FUNCTION_BLOCK "FB40_CommSlave"
{ S7_Optimized_Access := 'TRUE' }
VERSION : 0.1
   VAR_INPUT 
      InFromSlave { ExternalAccessible := 'False'; ExternalVisible := 'False'; ExternalWritable := 'False'} : "stSlaveToMaster";   // Communication data from slave PLC
      xDryRun { ExternalAccessible := 'False'; ExternalVisible := 'False'; ExternalWritable := 'False'} : Bool;   // Running in DryRun
      xResetGrafcet { ExternalAccessible := 'False'; ExternalVisible := 'False'; ExternalWritable := 'False'} : Bool;   // Reset robot communication grafcet in slave PLC
      xAutoMode { ExternalAccessible := 'False'; ExternalVisible := 'False'; ExternalWritable := 'False'} : Bool;   // Automatic mode
      xSemiAutoMode { ExternalAccessible := 'False'; ExternalVisible := 'False'; ExternalWritable := 'False'} : Bool;   // Semi-automatic mode
      xMaintenanceMode { ExternalAccessible := 'False'; ExternalVisible := 'False'; ExternalWritable := 'False'} : Bool;   // Maintenance mode
      xReset { ExternalAccessible := 'False'; ExternalVisible := 'False'; ExternalWritable := 'False'} : Bool;   // Command reset (Fault or safety)
      xPulseSeconde { ExternalAccessible := 'False'; ExternalVisible := 'False'; ExternalWritable := 'False'} : Bool;   // Bit 1 pulse each second
      xEnableStartRobot { ExternalAccessible := 'False'; ExternalVisible := 'False'; ExternalWritable := 'False'} : Bool;   // Operator Enable start robot
      xGlobalSafety { ExternalAccessible := 'False'; ExternalVisible := 'False'; ExternalWritable := 'False'} : Bool;   // Global safety srate of the cell
      xCbsDoorAccessClosed { ExternalAccessible := 'False'; ExternalVisible := 'False'; ExternalWritable := 'False'} : Bool;   // CBS door access closed
      xAccessReq { ExternalAccessible := 'False'; ExternalVisible := 'False'; ExternalWritable := 'False'} : Bool;   // Access requested to open the door
      xValideOperation { ExternalAccessible := 'False'; ExternalVisible := 'False'; ExternalWritable := 'False'} : Bool;   // Validation Operator to remove or Put disk on FerRobotic head
      xValideFault { ExternalAccessible := 'False'; ExternalVisible := 'False'; ExternalWritable := 'False'} : Bool;   // Validation Operator of Flatness fault
      xVaccumPumpRunning { ExternalAccessible := 'False'; ExternalVisible := 'False'; ExternalWritable := 'False'} : Bool;   // Vacuum Pump is running - zero speed detection
      xVacuumRunning { ExternalAccessible := 'False'; ExternalVisible := 'False'; ExternalWritable := 'False'} : Bool;   // Vacuum is running
      xOtherRobotHasStarted { ExternalAccessible := 'False'; ExternalVisible := 'False'; ExternalWritable := 'False'} : Bool;   // Robot on other side has started
      xOtherRobotFinished { ExternalAccessible := 'False'; ExternalVisible := 'False'; ExternalWritable := 'False'} : Bool;   // Robot on other side finished
      xBothRobotFinished { ExternalAccessible := 'False'; ExternalVisible := 'False'; ExternalWritable := 'False'} : Bool;   // Both robot finished
      xReqChangePaper { ExternalAccessible := 'False'; ExternalVisible := 'False'; ExternalWritable := 'False'} : Bool;   // Operator request changing paper
      xMaintStartProg { ExternalAccessible := 'False'; ExternalVisible := 'False'; ExternalWritable := 'False'} : Bool;   // Maintenance normal start
      xMaintStartMain { ExternalAccessible := 'False'; ExternalVisible := 'False'; ExternalWritable := 'False'} : Bool;   // Maintenance start main
      usiRawMaterial { ExternalAccessible := 'False'; ExternalVisible := 'False'; ExternalWritable := 'False'} : USInt;   // Raw materiel selected
      uiServicePathNum { ExternalAccessible := 'False'; ExternalVisible := 'False'; ExternalWritable := 'False'} : UInt;   // Service Path Number
      xParamManu { ExternalAccessible := 'False'; ExternalVisible := 'False'; ExternalWritable := 'False'} : "stFerRoboticParam";   // Manual parameter for FerRobotic Head
      xCmdManuLockGimball { ExternalAccessible := 'False'; ExternalVisible := 'False'; ExternalWritable := 'False'} : Bool;   // Manual command Lock Gimball
      xCmdManuLockEccentric1 { ExternalAccessible := 'False'; ExternalVisible := 'False'; ExternalWritable := 'False'} : Bool;   // Manual command Lock Eccentric 1
      xCmdManuLockEccentric2 { ExternalAccessible := 'False'; ExternalVisible := 'False'; ExternalWritable := 'False'} : Bool;   // Manual command Lock Eccentric 2
      xCmdManuLockEccentric3 { ExternalAccessible := 'False'; ExternalVisible := 'False'; ExternalWritable := 'False'} : Bool;   // Manual command Lock Eccentric 3
      xCmdManuEnableRotate { ExternalAccessible := 'False'; ExternalVisible := 'False'; ExternalWritable := 'False'} : Bool;   // Manual command Enable Rotation
      xCmdManuRemoveConfig { ExternalAccessible := 'False'; ExternalVisible := 'False'; ExternalWritable := 'False'} : Bool;   // Manual command for activate the Remove config on FerRobotic Head
      xCmdManuPickupConfig { ExternalAccessible := 'False'; ExternalVisible := 'False'; ExternalWritable := 'False'} : Bool;   // Manual command for activate the Pickup config on FerRobotic Head
      xCmdManuFlatnessConfig { ExternalAccessible := 'False'; ExternalVisible := 'False'; ExternalWritable := 'False'} : Bool;   // Manual command for activate the Flatness check config on FerRobotic Head
      xCmdManuOpenVacValve { ExternalAccessible := 'False'; ExternalVisible := 'False'; ExternalWritable := 'False'} : Bool;   // Manual commande to open Vacuum valve
      xCmdManuCloseVaValve { ExternalAccessible := 'False'; ExternalVisible := 'False'; ExternalWritable := 'False'} : Bool;   // Manual commande to close Vacuum valve
      xForceLubricationX { ExternalAccessible := 'False'; ExternalVisible := 'False'; ExternalWritable := 'False'} : Bool;   // Force to start greasing pump for X axis
      xForceLubricationZ { ExternalAccessible := 'False'; ExternalVisible := 'False'; ExternalWritable := 'False'} : Bool;   // Force to start greasing pump for Z axis
      xLightTest { ExternalAccessible := 'False'; ExternalVisible := 'False'; ExternalWritable := 'False'} : Bool;   // Command Light test
   END_VAR

   VAR_OUTPUT 
      OutToSlave { ExternalAccessible := 'False'; ExternalVisible := 'False'; ExternalWritable := 'False'} : "stMasterToSlave";   // Communication data to slave PLC
      xRobotInAuto { ExternalAccessible := 'False'; ExternalVisible := 'False'; ExternalWritable := 'False'} : Bool;   // Robot is automatic mode
      xRobotInManu { ExternalAccessible := 'False'; ExternalVisible := 'False'; ExternalWritable := 'False'} : Bool;   // Robot is in manual mode
      xRobotInHome { ExternalAccessible := 'False'; ExternalVisible := 'False'; ExternalWritable := 'False'} : Bool;   // Robot is in home position
      xRobotReqReset { ExternalAccessible := 'False'; ExternalVisible := 'False'; ExternalWritable := 'False'} : Bool;   // Robot request a reset command
      xRobotStopped { ExternalAccessible := 'False'; ExternalVisible := 'False'; ExternalWritable := 'False'} : Bool;   // Robot stopped
      xWarningStart { ExternalAccessible := 'False'; ExternalVisible := 'False'; ExternalWritable := 'False'} : Bool;   // Warning before start robot
      xReqVacuum { ExternalAccessible := 'False'; ExternalVisible := 'False'; ExternalWritable := 'False'} : Bool;   // Request enable vacuum
      xRecipeInProgress { ExternalAccessible := 'False'; ExternalVisible := 'False'; ExternalWritable := 'False'} : Bool;   // Sanding process is in progress
      xProductionRunning { ExternalAccessible := 'False'; ExternalVisible := 'False'; ExternalWritable := 'False'} : Bool;   // Production Running for Teep track
   END_VAR
   VAR_OUTPUT RETAIN
      xRobotHasStarted { ExternalAccessible := 'False'; ExternalVisible := 'False'; ExternalWritable := 'False'} : Bool;   // Robot has started
   END_VAR
   VAR_OUTPUT 
      xWaitOtherRobotFinished { ExternalAccessible := 'False'; ExternalVisible := 'False'; ExternalWritable := 'False'} : Bool;   // Wait robot on other side finished
      xWaitBothRobotFinished { ExternalAccessible := 'False'; ExternalVisible := 'False'; ExternalWritable := 'False'} : Bool;   // Wait both robot finished
      xMagazineEmpty { ExternalAccessible := 'False'; ExternalVisible := 'False'; ExternalWritable := 'False'} : Bool;
      xShowPopRemoveDisk { ExternalAccessible := 'False'; ExternalVisible := 'False'; ExternalWritable := 'False'} : Bool;
      xShowPopPickupDisk { ExternalAccessible := 'False'; ExternalVisible := 'False'; ExternalWritable := 'False'} : Bool;
      xShowPopFlatnessFault { ExternalAccessible := 'False'; ExternalVisible := 'False'; ExternalWritable := 'False'} : Bool;
      uiJobDataNumber { ExternalAccessible := 'False'; ExternalVisible := 'False'; ExternalWritable := 'False'} : UInt;   // Actual job data number
      xPathInProgress { ExternalAccessible := 'False'; ExternalVisible := 'False'; ExternalWritable := 'False'} : Bool;   // Service path in progress
      xPathStopped { ExternalAccessible := 'False'; ExternalVisible := 'False'; ExternalWritable := 'False'} : Bool;   // Service path stopped
      xPathCancelled { ExternalAccessible := 'False'; ExternalVisible := 'False'; ExternalWritable := 'False'} : Bool;   // Service path cancelled
      xContactState { ExternalAccessible := 'False'; ExternalVisible := 'False'; ExternalWritable := 'False'} : Bool;   // State of the FerRobotic head contact
      xVacValveOpen { ExternalAccessible := 'False'; ExternalVisible := 'False'; ExternalWritable := 'False'} : Bool;   // Vacuum valve open
      xVacValveClosed { ExternalAccessible := 'False'; ExternalVisible := 'False'; ExternalWritable := 'False'} : Bool;   // Vacuum valve close
      nActualForce { ExternalAccessible := 'False'; ExternalVisible := 'False'; ExternalWritable := 'False'} : Int;   // Actual force on FerRobotic head
      uiSetSpeed { ExternalAccessible := 'False'; ExternalVisible := 'False'; ExternalWritable := 'False'} : UInt;   // Speed set in Ferrobotic head
      uiRobotSpeed { ExternalAccessible := 'False'; ExternalVisible := 'False'; ExternalWritable := 'False'} : UInt;   // Speed set to the robot
      uiPaperChangeDistance { ExternalAccessible := 'False'; ExternalVisible := 'False'; ExternalWritable := 'False'} : UInt;
      rActualPosition { ExternalAccessible := 'False'; ExternalVisible := 'False'; ExternalWritable := 'False'} : Real;   // Actual position of the FerRobotic head
      xRangeFinderDetection { ExternalAccessible := 'False'; ExternalVisible := 'False'; ExternalWritable := 'False'} : Bool;
      uiRangeFinderValue { ExternalAccessible := 'False'; ExternalVisible := 'False'; ExternalWritable := 'False'} : UInt;
      uiCounterPulse_X { ExternalAccessible := 'False'; ExternalVisible := 'False'; ExternalWritable := 'False'} : UInt;
      uiCounterPulse_Z { ExternalAccessible := 'False'; ExternalVisible := 'False'; ExternalWritable := 'False'} : UInt;
      uiGreaseFault_X { ExternalAccessible := 'False'; ExternalVisible := 'False'; ExternalWritable := 'False'} : UInt;
      uiGreaseFault_Z { ExternalAccessible := 'False'; ExternalVisible := 'False'; ExternalWritable := 'False'} : UInt;
      uiDistanceSandingDisk { ExternalAccessible := 'False'; ExternalVisible := 'False'; ExternalWritable := 'False'} : UInt;
      uiActualRobotSpeed { ExternalAccessible := 'False'; ExternalVisible := 'False'; ExternalWritable := 'False'} : UInt;   // Actual speed of theTCP of the robot
      udiOdometer_X { ExternalAccessible := 'False'; ExternalVisible := 'False'; ExternalWritable := 'False'} : UDInt;
      udiOdometer_Z { ExternalAccessible := 'False'; ExternalVisible := 'False'; ExternalWritable := 'False'} : UDInt;
      uiDistanceBeforeGreasingX { ExternalAccessible := 'False'; ExternalVisible := 'False'; ExternalWritable := 'False'} : UInt;
      uiDistanceBeforeGreasingZ { ExternalAccessible := 'False'; ExternalVisible := 'False'; ExternalWritable := 'False'} : UInt;
      uiDiskUsed { ExternalAccessible := 'False'; ExternalVisible := 'False'; ExternalWritable := 'False'} : UInt;
      uiRobotStatus { ExternalAccessible := 'False'; ExternalVisible := 'False'; ExternalWritable := 'False'} : UInt;
      udiFaultTime { ExternalAccessible := 'False'; ExternalVisible := 'False'; ExternalWritable := 'False'} : UDInt;
      udiRunTime { ExternalAccessible := 'False'; ExternalVisible := 'False'; ExternalWritable := 'False'} : UDInt;
      udiPauseTime { ExternalAccessible := 'False'; ExternalVisible := 'False'; ExternalWritable := 'False'} : UDInt;
      udiRobotPowerOnTime { ExternalAccessible := 'False'; ExternalVisible := 'False'; ExternalWritable := 'False'} : UDInt;
      udiRobotDriveOnTime { ExternalAccessible := 'False'; ExternalVisible := 'False'; ExternalWritable := 'False'} : UDInt;
      bInput100 { ExternalAccessible := 'False'; ExternalVisible := 'False'; ExternalWritable := 'False'} : SInt;
      bInput101 { ExternalAccessible := 'False'; ExternalVisible := 'False'; ExternalWritable := 'False'} : SInt;
      bInput102 { ExternalAccessible := 'False'; ExternalVisible := 'False'; ExternalWritable := 'False'} : SInt;
      bInput103 { ExternalAccessible := 'False'; ExternalVisible := 'False'; ExternalWritable := 'False'} : SInt;
      bInputFast90 { ExternalAccessible := 'False'; ExternalVisible := 'False'; ExternalWritable := 'False'} : SInt;
      bInputSafety500 { ExternalAccessible := 'False'; ExternalVisible := 'False'; ExternalWritable := 'False'} : SInt;
      bOutput100 { ExternalAccessible := 'False'; ExternalVisible := 'False'; ExternalWritable := 'False'} : SInt;
      bOutput101 { ExternalAccessible := 'False'; ExternalVisible := 'False'; ExternalWritable := 'False'} : SInt;
      bOutputSafety508 { ExternalAccessible := 'False'; ExternalVisible := 'False'; ExternalWritable := 'False'} : SInt;
      nInput600 { ExternalAccessible := 'False'; ExternalVisible := 'False'; ExternalWritable := 'False'} : Int;
      nInput602 { ExternalAccessible := 'False'; ExternalVisible := 'False'; ExternalWritable := 'False'} : Int;
      nInput604 { ExternalAccessible := 'False'; ExternalVisible := 'False'; ExternalWritable := 'False'} : Int;
      nInput606 { ExternalAccessible := 'False'; ExternalVisible := 'False'; ExternalWritable := 'False'} : Int;
      wFaultFerRobotic { ExternalAccessible := 'False'; ExternalVisible := 'False'; ExternalWritable := 'False'} : Word;   // Fault on the FerRobotic head
      wFaultManageRobot { ExternalAccessible := 'False'; ExternalVisible := 'False'; ExternalWritable := 'False'} : Word;   // Fault on fonction management robot on the slave PLC
      wFaultRobot { ExternalAccessible := 'False'; ExternalVisible := 'False'; ExternalWritable := 'False'} : Word;   // Fault on the robot
      wFaultOther { ExternalAccessible := 'False'; ExternalVisible := 'False'; ExternalWritable := 'False'} : Word;
      wFaultVacuumValve { ExternalAccessible := 'False'; ExternalVisible := 'False'; ExternalWritable := 'False'} : Word;
      wFaultFerRoboticManage { ExternalAccessible := 'False'; ExternalVisible := 'False'; ExternalWritable := 'False'} : Word;
      wWarningDiskTrayEmpty { ExternalAccessible := 'False'; ExternalVisible := 'False'; ExternalWritable := 'False'} : Word;
   END_VAR

   VAR_IN_OUT 
      xStartRecipe { ExternalAccessible := 'False'; ExternalVisible := 'False'; ExternalWritable := 'False'} : Bool;   // Command start recipe selected
      xStopRecipe { ExternalAccessible := 'False'; ExternalVisible := 'False'; ExternalWritable := 'False'} : Bool;   // Command stop recipe in progress
      xCancelRecipe { ExternalAccessible := 'False'; ExternalVisible := 'False'; ExternalWritable := 'False'} : Bool;   // Command cancel Recipe in progress
      xStartSanding { ExternalAccessible := 'False'; ExternalVisible := 'False'; ExternalWritable := 'False'} : Bool;   // Start Sanding a new CBS
      xEndSanding { ExternalAccessible := 'False'; ExternalVisible := 'False'; ExternalWritable := 'False'} : Bool;   // End sanding
      xRobotUsed { ExternalAccessible := 'False'; ExternalVisible := 'False'; ExternalWritable := 'False'} : Bool;   // Robot was used for this CBS
      xStartPath { ExternalAccessible := 'False'; ExternalVisible := 'False'; ExternalWritable := 'False'} : Bool;   // Command start service path
      xStopPath { ExternalAccessible := 'False'; ExternalVisible := 'False'; ExternalWritable := 'False'} : Bool;   // Command stop service path
      xCancelPath { ExternalAccessible := 'False'; ExternalVisible := 'False'; ExternalWritable := 'False'} : Bool;   // Command Cancel service path
      usiSandingType { ExternalAccessible := 'False'; ExternalVisible := 'False'; ExternalWritable := 'False'} : USInt;   // Sanding type selected
      usiTrajNumber { ExternalAccessible := 'False'; ExternalVisible := 'False'; ExternalWritable := 'False'} : USInt;   // Robot trajectory number selected
      stFlatnessCtrlData : "stFlatnessData";
      aListJobData : Array[*] of "stJobData";   // Job Data list for current CBS program
   END_VAR

   VAR 
      sxMemStartRecipe { ExternalAccessible := 'False'; ExternalVisible := 'False'; ExternalWritable := 'False'} : Bool;
      sxMemPulse { ExternalAccessible := 'False'; ExternalVisible := 'False'; ExternalWritable := 'False'} : Bool;
      sxWarningFinished { ExternalAccessible := 'False'; ExternalVisible := 'False'; ExternalWritable := 'False'} : Bool;
      sxEnableWarning { ExternalAccessible := 'False'; ExternalVisible := 'False'; ExternalWritable := 'False'} : Bool;
   END_VAR
   VAR RETAIN
      sxMemNewCBS { ExternalAccessible := 'False'; ExternalVisible := 'False'; ExternalWritable := 'False'} : Bool;
      sxMemoryEndOfCBS { ExternalAccessible := 'False'; ExternalVisible := 'False'; ExternalWritable := 'False'} : Bool;
   END_VAR
   VAR 
      suiStep { ExternalAccessible := 'False'; ExternalVisible := 'False'; ExternalWritable := 'False'} : UInt;
      suiMaxJobNumber { ExternalAccessible := 'False'; ExternalVisible := 'False'; ExternalWritable := 'False'} : UInt;
      miDB_TonWarningStart {InstructionName := 'TON_TIME'; LibVersion := '1.0'; ExternalAccessible := 'False'; ExternalVisible := 'False'; ExternalWritable := 'False'} : TON_TIME;
      miDB_FPStartSanding {InstructionName := 'R_TRIG'; LibVersion := '1.0'; ExternalAccessible := 'False'; ExternalVisible := 'False'; ExternalWritable := 'False'} : R_TRIG;
      miDB_FPEndSanding {InstructionName := 'R_TRIG'; LibVersion := '1.0'; ExternalAccessible := 'False'; ExternalVisible := 'False'; ExternalWritable := 'False'} : R_TRIG;
   END_VAR

   VAR_TEMP 
      txFaultPresent : Bool;
      txEnableVacuum : Bool;
   END_VAR

   VAR CONSTANT 
      WaitSelectMode : UInt := 0;
      WaitStartRecipe : UInt := 10;
      WaitEndWarnStart : UInt := 20;
      WaitRecipeRunning : UInt := 30;
      RecipeRunning : UInt := 40;
      WaitRecipeStopped : UInt := 50;
      WaitReStartRecipe : UInt := 60;
      WaitDoorClosed : UInt := 70;
      WaitRecipeCancelled : UInt := 80;
      WaitOtherRobotFinished : UInt := 90;
      WaitBothRobotFinished : UInt := 95;
      WaitCarRemoved : UInt := 97;
      WaitStartPath : UInt := 100;
      WaitPathRunning : UInt := 110;
      PathRunning : UInt := 120;
      WaitPathCancelled : UInt := 130;
      PathCancelled : UInt := 135;
      WaitPathStopped : UInt := 140;
      PathStopped : UInt := 150;
      ManualMode : UInt := 200;
   END_VAR


BEGIN
	
	REGION Copy Robot Input
	  
	  // Fault and fult number
	  #wFaultFerRobotic := #InFromSlave.wFaultFerRobotic; // Fault number of FerRobot Head
	  #wFaultManageRobot := #InFromSlave.wFaultManageRobot; // Fault number in the robot management of the slave PLC
	  #wFaultRobot := #InFromSlave.wFaultRobot; // Fault number of the robot itself
	  #wFaultOther := #InFromSlave.wFaultOther; // Fault number of the greasing system axis X and Z
	  #wFaultVacuumValve := #InFromSlave.wFaultVacuumValve; // Fault number of Vacuum valve
	  #wFaultFerRoboticManage := #InFromSlave.wFaultFerRoboticManage; // Fault of FerRobotic management
	  #wWarningDiskTrayEmpty := #InFromSlave.wWarningDiskTrayEmpty; // Warning number
	  #txFaultPresent := (#wFaultFerRobotic <> 0) OR (#wFaultManageRobot <> 0) OR (#wFaultRobot <> 0) OR (#wFaultOther <> 0) OR (#wFaultVacuumValve <> 0) OR (#wFaultFerRoboticManage <> 0); // At least 1 fault is present
	  
	  // Display FerRobotic information
	  #nActualForce := #InFromSlave.nActualForce; // Actual force apply on the FerRobotic head in N
	  #rActualPosition := UINT_TO_REAL(#InFromSlave.uiActualPosition) / 10.0; // Actual position of th FerRobotic head in mm
	  #xContactState := (#InFromSlave.usiContact = 1); // Contact state between ferrobotic head and Carbody Shell
	  
	  // Robot stopped
	  #xRobotStopped := #InFromSlave.xRecipeStopped;
	  
	  // Robot in Home Position
	  #xRobotInHome := #InFromSlave.xRobotInHome;
	  
	  // Measure Laser State
	  #xRangeFinderDetection := #InFromSlave.xRangeFinder;
	  #uiRangeFinderValue := #InFromSlave.uiRangerFinder;
	  
	  // Greasing state
	  #uiCounterPulse_X := #InFromSlave.uiCounterPulse_X;
	  #uiCounterPulse_Z := #InFromSlave.uiCounterPulse_Z;
	  #uiGreaseFault_X := #InFromSlave.uiGreaseFault_X;
	  #uiGreaseFault_Z := #InFromSlave.uiGreaseFault_Z;
	  #uiDistanceSandingDisk := #InFromSlave.uiDistanceSandingDisk;
	  #uiActualRobotSpeed := #InFromSlave.uiActualRobotSpeed;
	  #udiOdometer_X := #InFromSlave.udiOdometer_X;
	  #udiOdometer_Z := #InFromSlave.udiOdometer_Z;
	  
	  // Show Popup state
	  #xShowPopFlatnessFault := #InFromSlave.xShowPopupFlatness;
	  #xShowPopPickupDisk := #InFromSlave.xShowPopupPickup;
	  #xShowPopRemoveDisk := #InFromSlave.xShowPopupRemove;
	  
	  //Time Robot
	  IF #xPulseSeconde AND (NOT #sxMemPulse) THEN
	    
	    #sxMemPulse := TRUE;
	    #udiFaultTime := #InFromSlave.udiFaultTime;
	    #udiRunTime := #InFromSlave.udiOperatingTime;
	    #udiPauseTime := #InFromSlave.udiPauseTime;
	    #udiRobotPowerOnTime := #InFromSlave.udiRobotPowerOn;
	    #udiRobotDriveOnTime := #InFromSlave.udiRobotDriveOn;
	    #uiDiskUsed := #InFromSlave.uiNbDisk;
	    
	  ELSIF (NOT #xPulseSeconde) AND #sxMemPulse THEN
	    #sxMemPulse := FALSE;
	  END_IF;
	  
	  #xMagazineEmpty := #InFromSlave.xMagazineEmpty;
	  
	  //Vacuum Valve State
	  #xVacValveOpen := #InFromSlave.xVacValveOpen;
	  #xVacValveClosed := #InFromSlave.xVacValveClosed;
	  
	  // Direct Input outut
	  #bInput100 := BYTE_TO_SINT(#InFromSlave.bInput100);
	  #bInput101 := BYTE_TO_SINT(#InFromSlave.bInput101);
	  #bInput102 := BYTE_TO_SINT(#InFromSlave.bInput102);
	  #bInput103 := BYTE_TO_SINT(#InFromSlave.bInput103);
	  #bInputFast90 := BYTE_TO_SINT(#InFromSlave.bInputFast90);
	  #bInputSafety500 := BYTE_TO_SINT(#InFromSlave.bInputSafety500);
	  #bOutput100 := BYTE_TO_SINT(#InFromSlave.bOutput100);
	  #bOutput101 := BYTE_TO_SINT(#InFromSlave.bOutput101);
	  #bOutputSafety508 := BYTE_TO_SINT(#InFromSlave.bOutputSafety508);
	  #nInput600 := #InFromSlave.nInput600;
	  #nInput602 := #InFromSlave.nInput602;
	  #nInput604 := #InFromSlave.nInput604;
	  #nInput606 := #InFromSlave.nInput606;
	  
	  // Flatness control
	  #stFlatnessCtrlData.xFlatnessCrtlRequestRecord := #InFromSlave.xReccordFlatness;
	  #stFlatnessCtrlData.xFlatnessCtrlPassed := #InFromSlave.xFlatnessDiskOk;
	  #stFlatnessCtrlData.uiStrokePositionDiskA := #InFromSlave.uiStrockPosDiskA;
	  #stFlatnessCtrlData.uiStrokePositionDiskB := #InFromSlave.uiStrockPosDiskB;
	  #stFlatnessCtrlData.uiStrokePositionDiskC := #InFromSlave.uiStrockPosDiskC;
	  
	END_REGION
	
	REGION Memory End Of CBS
	  
	  IF #InFromSlave.xRecipeEnded AND (NOT #sxMemoryEndOfCBS) THEN
	    #sxMemoryEndOfCBS := TRUE;
	  ELSIF (NOT #xCbsDoorAccessClosed) AND #sxMemoryEndOfCBS THEN
	    #sxMemoryEndOfCBS := FALSE;
	    #xRobotUsed := FALSE;
	  END_IF;
	    
	END_REGION
	REGION Mode management
	  // Select robot mode
	  IF #InFromSlave.xRobotInAuto AND (NOT #InFromSlave.xRobotInManu) THEN // Detection of robot operation mode
	    #xRobotInAuto := TRUE;
	    #xRobotInManu := FALSE;
	    //#OutToSlave.xManualMode := FALSE;
	  ELSE
	    #xRobotInAuto := FALSE;
	    #xRobotInManu := TRUE;
	    //#OutToSlave.xManualMode := TRUE;
	  END_IF;
	  
	  #OutToSlave.xManualMode := #xMaintenanceMode AND (#InFromSlave.xRobotInManu OR (NOT #InFromSlave.xRobotInAuto));
	  
	  // Prevent start robot if operator deseable it
	  IF (NOT #xEnableStartRobot) AND #xStartRecipe THEN
	    #xStartRecipe := FALSE;
	  END_IF;
	  
	  // Stop all if safety not ok
	  IF (NOT #xGlobalSafety)THEN
	    #suiStep := #WaitSelectMode;
	    #xStartRecipe := FALSE;
	    #xCancelRecipe := FALSE;
	    #xStopRecipe := FALSE;
	  ELSE
	    CASE #suiStep OF
	      #WaitSelectMode:  // Mode selection
	        IF #xAutoMode AND #xRobotInAuto THEN
	          #suiStep := #WaitStartRecipe;
	        ELSIF #xSemiAutoMode THEN
	          #suiStep := #WaitStartPath;
	        ELSIF #xMaintenanceMode AND #xRobotInManu THEN
	          #suiStep := #ManualMode;
	        END_IF;
	          
	        // ======================================================================================================  
	        // =========================Automatic mode===============================================================    
	      #WaitStartRecipe:
	        IF ((#OutToSlave.usiProgNumber <> 0) AND (#OutToSlave.usiLayerType <> 0)) AND #xStartRecipe AND (NOT #sxMemoryEndOfCBS) THEN
	          #suiStep := #WaitEndWarnStart;
	          #xStartRecipe := FALSE;
	        ELSIF #sxMemoryEndOfCBS THEN
	          #xStartRecipe := FALSE;
	          #suiStep := #WaitOtherRobotFinished;
	        ELSIF (NOT #xAutoMode) OR (NOT #xRobotInAuto) THEN
	          #xStartRecipe := FALSE;
	          #suiStep := #WaitSelectMode;
	        END_IF;
	          
	      #WaitEndWarnStart:
	        IF #xVacuumRunning AND #sxWarningFinished THEN
	          #suiStep := #WaitRecipeRunning;
	        END_IF;
	          
	      #WaitRecipeRunning:
	        IF #InFromSlave.xRecipeInProgress THEN
	          #suiStep := #RecipeRunning;
	        END_IF;
	          
	      #RecipeRunning:
	        IF #xStopRecipe THEN
	          #xStopRecipe := FALSE;
	          #suiStep := #WaitRecipeStopped;
	        ELSIF #xAccessReq THEN
	          #suiStep := #WaitDoorClosed;
	        ELSIF #xCancelRecipe THEN
	          #xCancelRecipe := FALSE;
	          #suiStep := #WaitRecipeCancelled;
	        ELSIF #InFromSlave.xRecipeEnded THEN
	          #suiStep := #WaitOtherRobotFinished;
	        ELSIF #InFromSlave.xRecipeWaitStart THEN
	          #suiStep := #WaitStartRecipe;
	        END_IF;
	
	      #WaitRecipeStopped:
	        IF #InFromSlave.xRecipeStopped THEN
	          #suiStep := #WaitReStartRecipe;
	        END_IF;
	        
	      #WaitReStartRecipe:
	        IF ((#OutToSlave.usiProgNumber <> 0) AND (#OutToSlave.usiLayerType <> 0)) AND #xStartRecipe THEN
	          #xStartRecipe := FALSE;
	          #suiStep := #WaitEndWarnStart;
	        END_IF;
	        
	      #WaitDoorClosed:
	        IF #InFromSlave.xRecipeStopped AND (NOT #xAccessReq) THEN
	          #suiStep := #WaitRecipeStopped;
	        END_IF;
	        
	      #WaitRecipeCancelled: // Wait for recipe finished
	        IF #InFromSlave.xRecipeEnded THEN
	          #suiStep := #WaitOtherRobotFinished;
	        END_IF;
	        
	      #WaitOtherRobotFinished: // Wait for other robot finish sanding or Other robot not started yet
	        IF #InFromSlave.xEndOfCBS AND (NOT #sxMemNewCBS) THEN
	          #sxMemNewCBS := TRUE;
	          #OutToSlave.xAckEndOfCBS := TRUE;
	        END_IF;
	        IF #xStartRecipe THEN
	          #xStartRecipe := FALSE;
	        END_IF;
	        IF (NOT #xOtherRobotHasStarted) OR #xOtherRobotFinished OR #xBothRobotFinished THEN
	          #xRobotUsed := TRUE;
	          #suiStep := #WaitBothRobotFinished;
	        END_IF;
	        
	      #WaitBothRobotFinished: // Wait Both robot finished or Other robot not started yet
	        IF (NOT #InFromSlave.xEndOfCBS) AND (NOT #xOtherRobotFinished) THEN
	          #suiStep := #WaitCarRemoved;
	        END_IF;
	        
	      #WaitCarRemoved:
	        IF (NOT #sxMemNewCBS) THEN
	          #suiStep := #WaitStartRecipe;
	        END_IF;
	        
	        // ======================================================================================================  
	        // =========================Semi-Automatic Mode==========================================================    
	      #WaitStartPath:
	        IF (#uiServicePathNum <> 0) AND #xStartPath THEN
	          #suiStep := #WaitPathRunning;
	        ELSIF (NOT #xSemiAutoMode) THEN
	          #suiStep := #WaitSelectMode;
	        END_IF;
	        
	      #WaitPathRunning:
	        IF #InFromSlave.xPathInProgress THEN
	          #suiStep := #PathRunning;
	        END_IF;
	        
	      #PathRunning:
	        IF #InFromSlave.xPathEnded THEN
	          #suiStep := #WaitStartPath;
	        ELSIF #xCancelPath OR (NOT #xSemiAutoMode) THEN
	          #suiStep := #WaitPathCancelled;
	        ELSIF #xStopPath THEN
	          #suiStep := #WaitPathStopped;
	        END_IF;
	        
	      #WaitPathCancelled:
	        IF #InFromSlave.xPathEnded THEN
	          #suiStep := #PathCancelled;
	        END_IF;
	        
	      #PathCancelled:
	        IF (NOT #xSemiAutoMode) THEN
	          #suiStep := #WaitSelectMode;
	        ELSE
	          #suiStep := #WaitStartPath;
	        END_IF;
	        
	      #WaitPathStopped:
	        IF #InFromSlave.xPathStopped THEN
	          #suiStep := #PathStopped;
	        END_IF;
	        
	      #PathStopped:
	        IF #xCancelPath THEN
	          #suiStep := #WaitPathCancelled;
	        ELSIF (NOT #xSemiAutoMode) THEN
	          #suiStep := #WaitSelectMode;
	        ELSIF ((#uiServicePathNum <> 0) AND (#uiServicePathNum = #InFromSlave.uiNumServicePath)) AND #xStartPath THEN
	          #suiStep := #WaitPathRunning;
	        END_IF;
	          
	        // ======================================================================================================  
	        // =========================Manual mode==================================================================    
	      #ManualMode:
	        IF (NOT #xMaintenanceMode) THEN
	          #suiStep := #WaitSelectMode;
	        END_IF;
	        
	      ELSE  // Statement section ELSE
	          ;
	    END_CASE;
	      
	  END_IF;
	    
	END_REGION
	
	REGION Manual Mode Management
	  IF (#suiStep = #ManualMode) THEN
	    #OutToSlave.ManualSandingPaperParam := #xParamManu; // FerRobotic parameter for manual mode
	    #OutToSlave.xCmdManuEnableRotate := #xCmdManuEnableRotate; // Enable sanding rotation
	    #OutToSlave.xCmdManuLockEccentric1 := #xCmdManuLockEccentric1; // Lock Eccentric 1
	    #OutToSlave.xCmdManuLockEccentric2 := #xCmdManuLockEccentric2; // Lock Eccentric 2
	    #OutToSlave.xCmdManuLockEccentric3 := #xCmdManuLockEccentric3; // Lock Eccentric 3
	    #OutToSlave.xCmdManuLockGimball := #xCmdManuLockGimball; // Lock Gimball
	    #OutToSlave.xCmdManuOpenVacValve := #xCmdManuOpenVacValve;
	    #OutToSlave.xCmdManuCloseVaValve := #xCmdManuCloseVaValve;
	    #OutToSlave.xCmdManuRemoveConfig := #xCmdManuRemoveConfig;
	    #OutToSlave.xCmdManuPickupConfig := #xCmdManuPickupConfig;
	    #OutToSlave.xCmdManuFlatnessConfig := #xCmdManuFlatnessConfig;
	  END_IF;
	END_REGION
	
	REGION Automatic Mode Management
	  
	  REGION Job Data Management
	    // Define the number max of reccord
	    #suiMaxJobNumber := DINT_TO_UINT(UPPER_BOUND(ARR := #aListJobData, DIM := 1));
	    // Select Job Data to send to the robot
	    IF (#InFromSlave.uiJobNumber > 0) AND (#InFromSlave.uiJobNumber <= #suiMaxJobNumber) THEN
	      #OutToSlave.JobData := #aListJobData[#InFromSlave.uiJobNumber];
	      #uiJobDataNumber := #InFromSlave.uiJobNumber;
	      #uiSetSpeed := #OutToSlave.JobData.SetSpeed;
	      #uiRobotSpeed := #OutToSlave.JobData.SetRobotSpeed;
	      #uiPaperChangeDistance := #OutToSlave.JobData.WornPaperDistance;
	      #OutToSlave.uiJobNumber := #InFromSlave.uiJobNumber;
	      #OutToSlave.xJobFound := TRUE;
	    ELSIF (#InFromSlave.uiJobNumber = 0) THEN
	      #OutToSlave.JobData := #aListJobData[0];
	      #uiJobDataNumber := #InFromSlave.uiJobNumber;
	      #uiSetSpeed := #OutToSlave.JobData.SetSpeed;
	      #uiRobotSpeed := #OutToSlave.JobData.SetRobotSpeed;
	      #OutToSlave.uiJobNumber := #InFromSlave.uiJobNumber;
	      #OutToSlave.xJobFound := FALSE;
	    ELSE
	      #OutToSlave.xJobFound := FALSE;
	    END_IF;
	  END_REGION
	  
	  REGION Warning Alarm
	    #sxEnableWarning := ((#suiStep = #WaitEndWarnStart) AND #xVacuumRunning AND #xVaccumPumpRunning);
	    #miDB_TonWarningStart(IN := #sxEnableWarning,
	                          PT := T#5S);
	    #sxWarningFinished := #miDB_TonWarningStart.Q;
	    #xWarningStart := #sxEnableWarning;
	  END_REGION
	  
	  #txEnableVacuum := (#suiStep = #WaitEndWarnStart) OR (#suiStep = #WaitRecipeRunning) OR (#suiStep = #RecipeRunning) OR (#suiStep = #WaitRecipeStopped) OR (#suiStep = #WaitDoorClosed) OR (#suiStep = #WaitRecipeCancelled);
	  #xReqVacuum := #txEnableVacuum;
	  
	  #xRecipeInProgress := (#suiStep = #RecipeRunning);
	  #xProductionRunning := (#suiStep = #WaitRecipeRunning) OR (#suiStep = #RecipeRunning) OR (#suiStep = #WaitRecipeStopped);
	  
	  // Reset commande Start, Stop or Cancel
	  IF (NOT #xRobotInAuto) OR (NOT #xAutoMode) THEN
	    #xStopRecipe := FALSE;
	    #xCancelRecipe := FALSE;
	    #xStartRecipe := FALSE;
	  ELSIF (#suiStep <> #RecipeRunning) THEN
	    #xStopRecipe := FALSE;
	  ELSIF (#suiStep <> #RecipeRunning)THEN
	    #xCancelRecipe := FALSE;
	  ELSIF ((#suiStep <> #WaitStartRecipe) AND (#suiStep <> #WaitReStartRecipe)) THEN
	    #xStartRecipe := FALSE;
	  END_IF;
	  
	  IF (#suiStep >= #WaitStartRecipe) AND (#suiStep <= #WaitOtherRobotFinished) THEN
	    #OutToSlave.usiProgNumber := #usiTrajNumber;
	    #OutToSlave.usiLayerType := #usiSandingType;
	  ELSE
	    #OutToSlave.usiProgNumber := #usiTrajNumber;
	    #OutToSlave.usiLayerType := #usiSandingType;
	  END_IF;
	  
	  // Communication inter robot
	  IF (#suiStep = #RecipeRunning) THEN
	    #xRobotHasStarted := TRUE;
	  ELSIF (#suiStep = #WaitOtherRobotFinished) THEN
	    #xRobotHasStarted := FALSE;
	  END_IF;
	  
	  #xWaitOtherRobotFinished := (#suiStep = #WaitOtherRobotFinished);
	  #xWaitBothRobotFinished := (#suiStep = #WaitBothRobotFinished);
	  
	  // Information Start sanding en End sanding
	  // for TipTrack and Production reccord
	  #miDB_FPStartSanding(CLK:=((#suiStep = #WaitEndWarnStart) AND #sxMemNewCBS));
	  IF #miDB_FPStartSanding.Q THEN
	    #xStartSanding := TRUE;
	  END_IF;
	  
	  #miDB_FPEndSanding(CLK:=(#suiStep = #WaitCarRemoved));
	  IF #miDB_FPEndSanding.Q THEN
	    #xEndSanding := TRUE;
	  END_IF;
	  
	END_REGION
	
	REGION Semi-Automatic mode management
	  
	  IF (#suiStep = #WaitStartPath) OR (#suiStep = #PathStopped) THEN
	    #OutToSlave.uiNumServicePath := #uiServicePathNum;
	  END_IF;
	  
	  #OutToSlave.xCancelPath := (#suiStep = #WaitPathCancelled);
	  #OutToSlave.xStartPath := (#suiStep = #WaitPathRunning);
	  #OutToSlave.xStopPath := (#suiStep = #WaitPathStopped);
	  
	  #xPathStopped := (#suiStep = #PathStopped);
	  #xPathInProgress := (#suiStep = #PathStopped);
	  #xPathCancelled := (#suiStep = #PathCancelled);
	  
	  IF (#suiStep <> #WaitStartPath) AND (#suiStep <> #PathStopped) THEN
	    #xStartPath := false;
	  ELSIF (#suiStep <> #PathRunning) THEN
	    #xStopPath := false;
	  ELSIF (#suiStep <> #PathRunning) AND (#suiStep <> #PathStopped) THEN
	    #xCancelPath := FALSE;
	  END_IF;
	  
	END_REGION
	
	REGION All Mode Management
	  
	  IF #xRobotInManu OR (NOT #xRobotInAuto) THEN
	    #uiRobotStatus := 0;  // Message robot In Manuel Mode
	  ELSIF #xRobotInAuto THEN
	    CASE #suiStep OF
	      #WaitEndWarnStart, #WaitRecipeRunning, #RecipeRunning:
	        #uiRobotStatus := 4; // Message robot Running
	        
	      #WaitReStartRecipe:
	        #uiRobotStatus := 3; // Message robot Paused
	        
	      #WaitOtherRobotFinished, #WaitBothRobotFinished, #WaitCarRemoved:
	        #uiRobotStatus := 2; // Message robot Stopped
	        
	      ELSE
	        #uiRobotStatus := 1; // Message robot In Automatic Mode
	        
	    END_CASE;
	  END_IF;
	  
	  #uiDistanceBeforeGreasingX := #InFromSlave.uiKmBeforeGresingX - #InFromSlave.uiCurrOdometerX;
	  #uiDistanceBeforeGreasingZ := #InFromSlave.uiKmBeforeGresingZ - #InFromSlave.uiCurrOdometerZ;
	  
	END_REGION
	
	REGION Copy robot output
	  
	  #OutToSlave.xReset := (#xReset AND (#InFromSlave.xResetReq OR (NOT #xGlobalSafety) OR #txFaultPresent)); // Send reset commande to the slave PLC
	  #OutToSlave.xGlobalSafety := #xGlobalSafety; // Send global safety state to the slave PLC
	  #OutToSlave.xAutoMode := #xAutoMode; // Automatic mode enable
	  #OutToSlave.xSemiAutoMode := #xSemiAutoMode; // Seim-Automatic mode enable
	  #OutToSlave.xMaintMode := #xMaintenanceMode; // Maintenance mode enable
	  #OutToSlave.xStartRobot := #xMaintStartProg; // Maintenance start program
	  #OutToSlave.xStartRobotMain := #xMaintStartMain; // Maintenance start main programm
	  #OutToSlave.xAccessReq := #xAccessReq; // Access in the the cell requested
	  #OutToSlave.xLightTest := #xLightTest; // Commande light test
	  #OutToSlave.xReqChangePaper := #xReqChangePaper; // Operator request changing disk
	  
	  #OutToSlave.xStartRecipe := (#suiStep = #WaitRecipeRunning);
	  #OutToSlave.xCancelRecipe := (#suiStep = #WaitRecipeCancelled);
	  #OutToSlave.xStopRecipe := (#suiStep = #WaitRecipeStopped) OR (#suiStep = #WaitDoorClosed);
	  #OutToSlave.xDryRun := #xDryRun;
	  #OutToSlave.xVacuumPumpRunning := #xVaccumPumpRunning;
	  
	  #OutToSlave.xStartUpWarning := #xWarningStart;
	  
	  #OutToSlave.xResetCounter := (#sxMemNewCBS AND #suiStep = #WaitEndWarnStart);
	  
	  IF #sxMemNewCBS AND #InFromSlave.xAckNewCBS THEN
	    #sxMemNewCBS := FALSE;
	  END_IF;
	  #OutToSlave.xNewCBS := #sxMemNewCBS;
	  
	  IF #OutToSlave.xAckEndOfCBS AND (NOT #InFromSlave.xEndOfCBS) THEN
	    #OutToSlave.xAckEndOfCBS := FALSE;
	  END_IF;
	  
	  
	  IF #xValideFault AND #InFromSlave.xShowPopupFlatness THEN
	    #OutToSlave.xValideFault := TRUE;
	  ELSIF #OutToSlave.xValideFault AND (NOT #InFromSlave.xShowPopupFlatness) THEN
	    #OutToSlave.xValideFault := FALSE;
	  END_IF;
	  
	  IF #xValideOperation AND (#InFromSlave.xShowPopupPickup OR #InFromSlave.xShowPopupRemove) THEN
	    #OutToSlave.xValideOperation := TRUE;
	  ELSIF #OutToSlave.xValideOperation AND (NOT #InFromSlave.xShowPopupPickup) AND (NOT #InFromSlave.xShowPopupRemove) THEN
	    #OutToSlave.xValideOperation := FALSE;
	  END_IF;
	  
	  // Flatness control
	  #OutToSlave.xAckReccordFlatness := #stFlatnessCtrlData.xFlatnessCtrlRecorded;
	  
	  // Force greasing axis
	  #OutToSlave.xForceLubricationX := #xForceLubricationX;
	  #OutToSlave.xForceLubricationZ := #xForceLubricationZ;
	  
	  // Reset grafcet of Robot communication
	  #OutToSlave.xResetGR7 := #xResetGrafcet;
	END_REGION
END_FUNCTION_BLOCK

FUNCTION "FC50_RecipeManage" : Void   // FC50, LAD
{ S7_Optimized_Access := 'TRUE' }
// stored: AutoNumber false, IsIECCheckEnabled true, SetENOAutomatically false
BEGIN

REGION Network 1: Management of recipde (Load, Save, Creat )
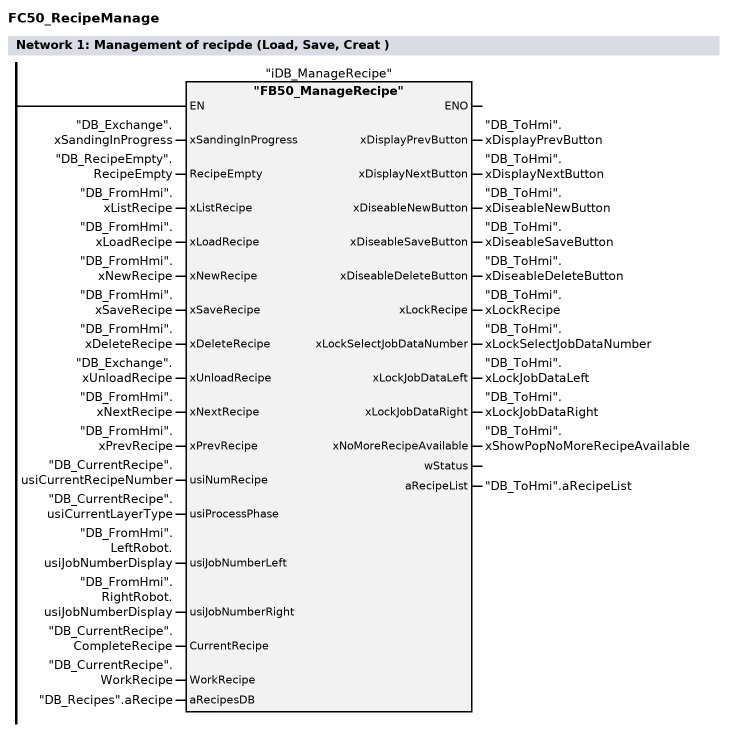
   RUNG wire#powerrail
      "iDB_ManageRecipe"(xSandingInProgress := "DB_Exchange".xSandingInProgress, RecipeEmpty := "DB_RecipeEmpty".RecipeEmpty, xListRecipe := "DB_FromHmi".xListRecipe, xLoadRecipe := "DB_FromHmi".xLoadRecipe, xNewRecipe := "DB_FromHmi".xNewRecipe, xSaveRecipe := "DB_FromHmi".xSaveRecipe, xDeleteRecipe := "DB_FromHmi".xDeleteRecipe, xUnloadRecipe := "DB_Exchange".xUnloadRecipe, xNextRecipe := "DB_FromHmi".xNextRecipe, xPrevRecipe := "DB_FromHmi".xPrevRecipe, usiNumRecipe := "DB_CurrentRecipe".usiCurrentRecipeNumber, usiProcessPhase := "DB_CurrentRecipe".usiCurrentLayerType, usiJobNumberLeft := "DB_FromHmi".LeftRobot.usiJobNumberDisplay, usiJobNumberRight := "DB_FromHmi".RightRobot.usiJobNumberDisplay, CurrentRecipe := "DB_CurrentRecipe".CompleteRecipe, WorkRecipe := "DB_CurrentRecipe".WorkRecipe, aRecipesDB := "DB_Recipes".aRecipe, xDisplayPrevButton => "DB_ToHmi".xDisplayPrevButton, xDisplayNextButton => "DB_ToHmi".xDisplayNextButton, xDiseableNewButton => "DB_ToHmi".xDiseableNewButton, xDiseableSaveButton => "DB_ToHmi".xDiseableSaveButton, xDiseableDeleteButton => "DB_ToHmi".xDiseableDeleteButton, xLockRecipe => "DB_ToHmi".xLockRecipe, xLockSelectJobDataNumber => "DB_ToHmi".xLockSelectJobDataNumber, xLockJobDataLeft => "DB_ToHmi".xLockJobDataLeft, xLockJobDataRight => "DB_ToHmi".xLockJobDataRight, xNoMoreRecipeAvailable => "DB_ToHmi".xShowPopNoMoreRecipeAvailable, wStatus =>, aRecipeList => "DB_ToHmi".aRecipeList)
   END_RUNG
   // the same network as SCL:
   "iDB_ManageRecipe"(xSandingInProgress := "DB_Exchange".xSandingInProgress,   // "FB50_ManageRecipe"
                      RecipeEmpty := "DB_RecipeEmpty".RecipeEmpty,
                      xListRecipe := "DB_FromHmi".xListRecipe,
                      xLoadRecipe := "DB_FromHmi".xLoadRecipe,
                      xNewRecipe := "DB_FromHmi".xNewRecipe,
                      xSaveRecipe := "DB_FromHmi".xSaveRecipe,
                      xDeleteRecipe := "DB_FromHmi".xDeleteRecipe,
                      xUnloadRecipe := "DB_Exchange".xUnloadRecipe,
                      xNextRecipe := "DB_FromHmi".xNextRecipe,
                      xPrevRecipe := "DB_FromHmi".xPrevRecipe,
                      usiNumRecipe := "DB_CurrentRecipe".usiCurrentRecipeNumber,
                      usiProcessPhase := "DB_CurrentRecipe".usiCurrentLayerType,
                      usiJobNumberLeft := "DB_FromHmi".LeftRobot.usiJobNumberDisplay,
                      usiJobNumberRight := "DB_FromHmi".RightRobot.usiJobNumberDisplay,
                      CurrentRecipe := "DB_CurrentRecipe".CompleteRecipe,
                      WorkRecipe := "DB_CurrentRecipe".WorkRecipe,
                      aRecipesDB := "DB_Recipes".aRecipe,
                      xDisplayPrevButton => "DB_ToHmi".xDisplayPrevButton,
                      xDisplayNextButton => "DB_ToHmi".xDisplayNextButton,
                      xDiseableNewButton => "DB_ToHmi".xDiseableNewButton,
                      xDiseableSaveButton => "DB_ToHmi".xDiseableSaveButton,
                      xDiseableDeleteButton => "DB_ToHmi".xDiseableDeleteButton,
                      xLockRecipe => "DB_ToHmi".xLockRecipe,
                      xLockSelectJobDataNumber => "DB_ToHmi".xLockSelectJobDataNumber,
                      xLockJobDataLeft => "DB_ToHmi".xLockJobDataLeft,
                      xLockJobDataRight => "DB_ToHmi".xLockJobDataRight,
                      xNoMoreRecipeAvailable => "DB_ToHmi".xShowPopNoMoreRecipeAvailable,
                      aRecipeList => "DB_ToHmi".aRecipeList);
END_REGION
END_FUNCTION

FUNCTION_BLOCK "FB50_ManageRecipe"
{ S7_Optimized_Access := 'TRUE' }
VERSION : 0.1
   VAR_INPUT 
      xSandingInProgress { ExternalAccessible := 'False'; ExternalVisible := 'False'; ExternalWritable := 'False'} : Bool;   // Sanding process is in progress
      RecipeEmpty { ExternalAccessible := 'False'; ExternalVisible := 'False'; ExternalWritable := 'False'} : "stRecipe";   // Recipe empty for delete the curent recipe data
   END_VAR

   VAR_OUTPUT 
      xDisplayPrevButton { ExternalAccessible := 'False'; ExternalVisible := 'False'; ExternalWritable := 'False'} : Bool;   // Display previous button in recipe screen
      xDisplayNextButton { ExternalAccessible := 'False'; ExternalVisible := 'False'; ExternalWritable := 'False'} : Bool;   // Display next button in recipe screen
      xDiseableNewButton { ExternalAccessible := 'False'; ExternalVisible := 'False'; ExternalWritable := 'False'} : Bool;   // Diseable new recipe button
      xDiseableSaveButton { ExternalAccessible := 'False'; ExternalVisible := 'False'; ExternalWritable := 'False'} : Bool;   // Diseable save recipe button
      xDiseableDeleteButton { ExternalAccessible := 'False'; ExternalVisible := 'False'; ExternalWritable := 'False'} : Bool;   // Diseable delete recipe button
      xLockRecipe { ExternalAccessible := 'False'; ExternalVisible := 'False'; ExternalWritable := 'False'} : Bool;   // Lock Modification recipe
      xLockSelectJobDataNumber { ExternalAccessible := 'False'; ExternalVisible := 'False'; ExternalWritable := 'False'} : Bool;   // Lock selection of job data number
      xLockJobDataLeft { ExternalAccessible := 'False'; ExternalVisible := 'False'; ExternalWritable := 'False'} : Bool;   // Lock modification Job Data left robot
      xLockJobDataRight { ExternalAccessible := 'False'; ExternalVisible := 'False'; ExternalWritable := 'False'} : Bool;   // Lock modification Job Data right robot
      xNoMoreRecipeAvailable { ExternalAccessible := 'False'; ExternalVisible := 'False'; ExternalWritable := 'False'} : Bool;   // No free recipe are available
      wStatus { ExternalAccessible := 'False'; ExternalVisible := 'False'; ExternalWritable := 'False'} : Word;   // Status word for debug
      aRecipeList { ExternalAccessible := 'False'; ExternalVisible := 'False'; ExternalWritable := 'False'} : Array[1..10] of "stRecipeListHMI";   // List of the recipe name display on HMI
   END_VAR

   VAR_IN_OUT 
      xListRecipe { ExternalAccessible := 'False'; ExternalVisible := 'False'; ExternalWritable := 'False'} : Bool;   // Make the list of all available recipe in the data base
      xLoadRecipe { ExternalAccessible := 'False'; ExternalVisible := 'False'; ExternalWritable := 'False'} : Bool;   // Load the recipe from the data base
      xNewRecipe { ExternalAccessible := 'False'; ExternalVisible := 'False'; ExternalWritable := 'False'} : Bool;   // Search for the next recipe free
      xSaveRecipe { ExternalAccessible := 'False'; ExternalVisible := 'False'; ExternalWritable := 'False'} : Bool;   // Save the current recipe in the data base
      xDeleteRecipe { ExternalAccessible := 'False'; ExternalVisible := 'False'; ExternalWritable := 'False'} : Bool;   // Delecte current recipe from data base
      xUnloadRecipe { ExternalAccessible := 'False'; ExternalVisible := 'False'; ExternalWritable := 'False'} : Bool;   // Unload current recipe
      xNextRecipe { ExternalAccessible := 'False'; ExternalVisible := 'False'; ExternalWritable := 'False'} : Bool;   // Load next Recipe in the Recipes list
      xPrevRecipe { ExternalAccessible := 'False'; ExternalVisible := 'False'; ExternalWritable := 'False'} : Bool;   // Load previous Recipe in the Recipes list
      usiNumRecipe { ExternalAccessible := 'False'; ExternalVisible := 'False'; ExternalWritable := 'False'} : USInt;   // Number of the current recipe
      usiProcessPhase { ExternalAccessible := 'False'; ExternalVisible := 'False'; ExternalWritable := 'False'} : USInt;
      usiJobNumberLeft { ExternalAccessible := 'False'; ExternalVisible := 'False'; ExternalWritable := 'False'} : USInt;   // Job number required by left robot
      usiJobNumberRight { ExternalAccessible := 'False'; ExternalVisible := 'False'; ExternalWritable := 'False'} : USInt;   // Job number required by right robot
      CurrentRecipe : "stRecipe";   // Current recipe
      WorkRecipe : "stWorkRecipe";
      aRecipesDB : Array[0..256] of "stRecipe";   // Data base of the recipe
   END_VAR

   VAR 
      sxRecipeLoaded { ExternalAccessible := 'False'; ExternalVisible := 'False'; ExternalWritable := 'False'} : Bool;
      sxRecipeSaved { ExternalAccessible := 'False'; ExternalVisible := 'False'; ExternalWritable := 'False'} : Bool;
      sxReadDblBusy { ExternalAccessible := 'False'; ExternalVisible := 'False'; ExternalWritable := 'False'} : Bool;
      sxListDblBusy { ExternalAccessible := 'False'; ExternalVisible := 'False'; ExternalWritable := 'False'} : Bool;
      sxWriteDblBusy { ExternalAccessible := 'False'; ExternalVisible := 'False'; ExternalWritable := 'False'} : Bool;
      sxListRecipe { ExternalAccessible := 'False'; ExternalVisible := 'False'; ExternalWritable := 'False'} : Bool;
      sxOperationInProgress { ExternalAccessible := 'False'; ExternalVisible := 'False'; ExternalWritable := 'False'} : Bool;   // Operation in progress
      sxUpdateDisplayList { ExternalAccessible := 'False'; ExternalVisible := 'False'; ExternalWritable := 'False'} : Bool;
      sxRecipeSelectFound { ExternalAccessible := 'False'; ExternalVisible := 'False'; ExternalWritable := 'False'} : Bool;
      snReadDblResult { ExternalAccessible := 'False'; ExternalVisible := 'False'; ExternalWritable := 'False'} : Int;
      snWriteDblResult { ExternalAccessible := 'False'; ExternalVisible := 'False'; ExternalWritable := 'False'} : Int;
      snListDblResult { ExternalAccessible := 'False'; ExternalVisible := 'False'; ExternalWritable := 'False'} : Int;
      suiStepLoadRecipe { ExternalAccessible := 'False'; ExternalVisible := 'False'; ExternalWritable := 'False'} : UInt;
      suiStepSaveRecipe { ExternalAccessible := 'False'; ExternalVisible := 'False'; ExternalWritable := 'False'} : UInt;
      suiStepListRecipe { ExternalAccessible := 'False'; ExternalVisible := 'False'; ExternalWritable := 'False'} : UInt;
      suicount { ExternalAccessible := 'False'; ExternalVisible := 'False'; ExternalWritable := 'False'} : UInt;
      suiCurrentIndexRecipe { ExternalAccessible := 'False'; ExternalVisible := 'False'; ExternalWritable := 'False'} : UInt;
      suiNextRecipeFree { ExternalAccessible := 'False'; ExternalVisible := 'False'; ExternalWritable := 'False'} : UInt;
      suiTotalOfRecipe { ExternalAccessible := 'False'; ExternalVisible := 'False'; ExternalWritable := 'False'} : UInt;
      suiIndexDisplay { ExternalAccessible := 'False'; ExternalVisible := 'False'; ExternalWritable := 'False'} : UInt;
      suiMemIndexDisplay { ExternalAccessible := 'False'; ExternalVisible := 'False'; ExternalWritable := 'False'} : UInt;
      suiCount_1 { ExternalAccessible := 'False'; ExternalVisible := 'False'; ExternalWritable := 'False'} : UInt;
      susiCurrentIndexList { ExternalAccessible := 'False'; ExternalVisible := 'False'; ExternalWritable := 'False'} : USInt;
      susiMemProcessPhase { ExternalAccessible := 'False'; ExternalVisible := 'False'; ExternalWritable := 'False'} : USInt;
      TempRecipe { ExternalAccessible := 'False'; ExternalVisible := 'False'; ExternalWritable := 'False'; S7_SetPoint := 'False'} : "stRecipe";
      aListRecipe { ExternalAccessible := 'False'; ExternalVisible := 'False'; ExternalWritable := 'False'; S7_SetPoint := 'False'} : Array[1..255] of "stItemListRecipe";   // List of recipe available in the data base
      miDB_FPLockSelectRecipe {InstructionName := 'R_TRIG'; LibVersion := '1.0'; ExternalAccessible := 'False'; ExternalVisible := 'False'; ExternalWritable := 'False'; S7_SetPoint := 'False'} : R_TRIG;
      miDB_FNLockSelectRecipe {InstructionName := 'F_TRIG'; LibVersion := '1.0'; ExternalAccessible := 'False'; ExternalVisible := 'False'; ExternalWritable := 'False'; S7_SetPoint := 'False'} : F_TRIG;
      suiCountLock : UInt;
      suiLastRecipe { ExternalAccessible := 'False'; ExternalVisible := 'False'; ExternalWritable := 'False'} : UInt;
      susiMaxLoad { ExternalAccessible := 'False'; ExternalVisible := 'False'; ExternalWritable := 'False'} : USInt;
   END_VAR

   VAR_TEMP 
      txReqReadRecipe : Bool;
      txReqWriteRecipe : Bool;
      txReqListRecipe : Bool;
   END_VAR

   VAR CONSTANT 
      stepCtrlRecipeNumber : UInt := 0;
      stepStartLoadRecipe : UInt := 10;
      stepLoadRecipe : UInt := 20;
      stepLoadRecipeCompleted : UInt := 30;
      stepLoadCompleted : UInt := 40;
      stepStartSaveRecipe : UInt := 10;
      stepSaveRecipe : UInt := 20;
      stepSaveRecipeCompleted : UInt := 30;
      stepSaveCompleted : UInt := 40;
      stepInitList : UInt := 0;
      stepCtrlListRecipeNumber : UInt := 10;
      stepStartListLoadRecipe : UInt := 20;
      stepListLoadRecipe : UInt := 30;
      StepListWaitOneCycle : UInt := 35;
      stepListLoadCompleted : UInt := 40;
   END_VAR


BEGIN
	// Force to make the list of recipe before load the recipe
	IF (NOT #sxRecipeLoaded) AND (#suiNextRecipeFree = 0) AND (NOT #sxListRecipe) THEN // Load the list of recipe before load the recipe
	  
	  REGION Force List recipe before load recipe
	    #sxListRecipe := TRUE;
	    #suiStepListRecipe := #stepInitList;
	  END_REGION
	  
	  // Load recipe from DB_Recipes in the load mmemory of the PLC to the DB_CurrentRecipe
	ELSIF (NOT #sxRecipeLoaded) AND (#suiNextRecipeFree <> 0) AND (NOT #sxListRecipe) THEN
	  
	  REGION Load recipe
	    #sxOperationInProgress := TRUE;
	    #sxRecipeSaved := TRUE;
	    CASE #suiStepLoadRecipe OF
	      #stepCtrlRecipeNumber: // Control if the Recipe Number is in range of 1 to 255
	        IF (#usiNumRecipe = 0) AND (#suiTotalOfRecipe = 0) THEN // No recipe loaded before and no recipe in the data base
	          #usiNumRecipe := 1;
	        ELSIF (#usiNumRecipe = 0) AND (#suiTotalOfRecipe <> 0) THEN // No recipe loaded before and less then one recipe listed in the data base
	          #usiNumRecipe := UINT_TO_USINT(#aListRecipe[1].RecipeIndex);
	        ELSIF #usiNumRecipe > 255 THEN
	          #usiNumRecipe := 255;
	        END_IF;
	        #suiStepLoadRecipe := #stepStartLoadRecipe;
	        
	      #stepStartLoadRecipe: // Start to read the source DB to put the recipe in the destination DB
	        IF (#snReadDblResult = 16#7002) THEN // Reading is in progress
	          #suiStepLoadRecipe := #stepLoadRecipe;
	        ELSIF (#snReadDblResult > 16#8000) THEN // Reading Error
	          #wStatus := INT_TO_WORD(#snReadDblResult);
	        END_IF;
	        
	      #stepLoadRecipe: // Waiting for reading completed
	        IF (NOT #sxReadDblBusy) THEN
	          #WorkRecipe.RecipeName := #CurrentRecipe.RecipeName;
	          #WorkRecipe.RecipeCbsType := #CurrentRecipe.RecipeCbsType;
	          #WorkRecipe.RecipeRawMaterial := #CurrentRecipe.RecipeRawMaterial;
	          #WorkRecipe.RecipeTrajNumber := #CurrentRecipe.RecipeTrajNumber;
	          #WorkRecipe.RecipeLayerType.JobTableLeft[0] := #RecipeEmpty.RecipeLayerType[1].JobTableLeft[0];
	          #WorkRecipe.RecipeLayerType.JobTableRight[0] := #RecipeEmpty.RecipeLayerType[1].JobTableRight[0];
	          #usiJobNumberLeft := 0;
	          #usiJobNumberRight := 0;
	          #usiProcessPhase := 0;
	          #sxUpdateDisplayList := TRUE;
	          #sxRecipeLoaded := TRUE;
	          #suiStepLoadRecipe := #stepLoadCompleted;
	        END_IF;
	        
	      #stepLoadCompleted:
	        ;// Do nothing
	      ELSE
	        ;// Normali case not possible
	    END_CASE;
	  END_REGION
	  
	  // Save the DB_CurrentRecipe in the DB_Recipes in the load mmemory of the PLC
	ELSIF (NOT #sxRecipeSaved) AND (NOT #sxListRecipe) THEN
	  
	  REGION Save recipe
	    #sxOperationInProgress := TRUE;
	    #sxRecipeLoaded := TRUE;
	    CASE #suiStepSaveRecipe OF
	      #stepCtrlRecipeNumber: // Control if the REcipe Number is in range of 1 to 255
	        IF #usiNumRecipe = 0 THEN
	          #usiNumRecipe := 1;
	        ELSIF #usiNumRecipe > 255 THEN
	          #usiNumRecipe := 255;
	        END_IF;
	        #CurrentRecipe.RecipeName := #WorkRecipe.RecipeName;
	        #CurrentRecipe.RecipeCbsType := #WorkRecipe.RecipeCbsType;
	        #CurrentRecipe.RecipeRawMaterial := #WorkRecipe.RecipeRawMaterial;
	        #CurrentRecipe.RecipeTrajNumber := #WorkRecipe.RecipeTrajNumber;
	        IF (#usiProcessPhase = 1) OR (#usiProcessPhase = 2) THEN
	          #CurrentRecipe.RecipeLayerType[#usiProcessPhase] := #WorkRecipe.RecipeLayerType;
	        END_IF;
	        #suiStepSaveRecipe := #stepStartSaveRecipe;
	        
	      #stepStartSaveRecipe: // Start to write the source DB to put the recipe in the destination DB
	        IF (#snWriteDblResult = 16#7002) THEN // Writing is in progress
	          #suiStepSaveRecipe := #stepSaveRecipe;
	        ELSIF (#snWriteDblResult > 16#8000) THEN // Reading Error
	          #wStatus := INT_TO_WORD(#snReadDblResult);
	        END_IF;
	        
	      #stepSaveRecipe: // Waiting for wrinting completed
	        IF (NOT #sxWriteDblBusy) THEN
	          #sxRecipeSaved := TRUE;
	          #sxListRecipe := TRUE;
	          #suiStepListRecipe := #stepInitList;
	          #suiStepSaveRecipe := #stepSaveCompleted;
	        END_IF;
	        
	      #stepSaveCompleted:
	        ;// Do nothing
	      ELSE
	        ;// Normali case not possible
	    END_CASE;
	  END_REGION
	  
	  // Make the list of all the recipe in the data base
	ELSIF #sxListRecipe THEN
	  
	  REGION Load list of recipe
	    #sxOperationInProgress := TRUE;
	    CASE #suiStepListRecipe OF
	      #stepInitList: // Initialise the Recipe list and the indexs
	        FOR #suicount := 1 TO 255 DO
	          #aListRecipe[#suicount].RecipeIndex := 0;
	          #aListRecipe[#suicount].RecipeName := '';
	        END_FOR;
	        #suiTotalOfRecipe := 0;
	        #suiNextRecipeFree := 999;
	        #susiCurrentIndexList := 0;
	        #suiCurrentIndexRecipe := 0;
	        #sxRecipeSelectFound := FALSE;
	        IF #suiLastRecipe = 0 THEN
	          #susiMaxLoad := 255;
	        ELSE
	          #susiMaxLoad := UINT_TO_USINT(#suiLastRecipe) + 2;
	          IF #susiMaxLoad > 255 THEN
	            #susiMaxLoad := 255;
	          END_IF;
	        END_IF;
	        #suiStepListRecipe := #stepCtrlListRecipeNumber;
	        
	      #stepCtrlListRecipeNumber: // Control if the Recipe Number is in range of 1 to 255
	        IF #susiCurrentIndexList < #susiMaxLoad THEN // Not all the recipe in the data base are read
	          #susiCurrentIndexList += 1;
	          #suiStepListRecipe := #stepStartListLoadRecipe;
	        ELSE // All the recipe in the datra base are read
	          IF (NOT #sxRecipeSelectFound) THEN
	            #usiNumRecipe := 0;
	            #usiJobNumberLeft := 0;
	            #usiJobNumberRight := 0;
	            #usiProcessPhase := 0;
	          END_IF;
	          #sxListRecipe := FALSE;
	          #sxUpdateDisplayList := TRUE;
	          #suiStepListRecipe := #stepListLoadCompleted;
	        END_IF;
	        
	      #stepStartListLoadRecipe: // Start to read the source DB to put the recipe in the destination DB
	        IF (#snListDblResult = 16#7002) THEN // Reading is in progress
	          #suiStepListRecipe := #stepListLoadRecipe;
	        ELSIF (#snListDblResult > 16#8000) THEN // Reading Error
	          #wStatus := INT_TO_WORD(#snListDblResult);
	        END_IF;
	        
	      #stepListLoadRecipe: // Waiting for reading completed
	        IF (NOT #sxReadDblBusy) AND  (#snListDblResult = 16#7000) AND (#TempRecipe.RecipeName <> '') THEN // Recipe recorded in the data base
	          #suiCurrentIndexRecipe += 1;
	          #suiTotalOfRecipe += 1;
	          #aListRecipe[#suiCurrentIndexRecipe].RecipeIndex := #susiCurrentIndexList;
	          #aListRecipe[#suiCurrentIndexRecipe].RecipeName := #TempRecipe.RecipeName;
	          IF (#susiCurrentIndexList = #usiNumRecipe) THEN
	            #sxRecipeSelectFound := TRUE;
	          END_IF;
	          #suiStepListRecipe := #StepListWaitOneCycle;
	        ELSIF (NOT #sxReadDblBusy) AND  (#snListDblResult = 16#7000) AND (#TempRecipe.RecipeName = '') THEN // No recipe recorded in the data base
	          IF (#suiNextRecipeFree = 999) THEN
	            #xNoMoreRecipeAvailable := FALSE;
	            #suiNextRecipeFree := #susiCurrentIndexList;
	          END_IF;
	          #suiStepListRecipe := #StepListWaitOneCycle;
	        END_IF;
	        
	      #StepListWaitOneCycle:
	        IF (#snListDblResult = 16#7000) OR (#snListDblResult = 16#0) THEN
	          #suiStepListRecipe := #stepCtrlListRecipeNumber;
	          #suiLastRecipe := #suiCurrentIndexRecipe;
	        END_IF;
	        
	      #stepListLoadCompleted: // list OF recipe available completed
	        ;// Do nothing
	        
	      ELSE
	        ;// Normali case not possible
	    END_CASE;
	  END_REGION
	  
	  // Waiting Operator request
	ELSIF (#sxRecipeLoaded AND #sxRecipeSaved AND (NOT #sxListRecipe)) THEN
	  
	  REGION Waiting command Load, Save, New, List or Delecte
	    #sxOperationInProgress := FALSE;
	    IF #xListRecipe THEN // User press List Recipe
	      #sxOperationInProgress := TRUE;
	      #xListRecipe := FALSE;
	      #suiStepListRecipe := #stepInitList;
	      #sxListRecipe := TRUE;
	      
	    ELSIF #xLoadRecipe THEN // User Press load recipe
	      #sxOperationInProgress := TRUE;
	      #xLoadRecipe := FALSE;
	      #suiStepLoadRecipe := #stepCtrlRecipeNumber;
	      #sxRecipeLoaded := FALSE;
	      
	    ELSIF #xNewRecipe THEN // User press new free recipe
	      #xNewRecipe := FALSE;
	      IF #suiNextRecipeFree <> 0 THEN
	        #sxOperationInProgress := TRUE;
	        #usiNumRecipe := UINT_TO_USINT(#suiNextRecipeFree); // Select the first free recipe
	        FOR #suicount := 1 TO 255 DO // Search first free display recipe
	          IF #aListRecipe[#suicount].RecipeName = '' THEN
	            #aListRecipe[#suicount].RecipeName := 'New'; // Create a temporari name for display in the list
	            #aListRecipe[#suicount].RecipeIndex := #usiNumRecipe; // Create a temporari index for display in the list
	            EXIT; // exit of the for loop
	          END_IF;
	        END_FOR;
	        #suiIndexDisplay := ((((#suicount - 1) / 10) * 10) + 1); // select the new display index
	        #sxUpdateDisplayList := TRUE; // request update the list
	        #suiStepLoadRecipe := #stepCtrlRecipeNumber;
	        #sxRecipeLoaded := FALSE;
	      ELSE
	        // No more recipe available
	        #xNoMoreRecipeAvailable := TRUE;
	      END_IF;
	      
	    ELSIF #xSaveRecipe THEN  // User press Save recipe
	      #sxOperationInProgress := TRUE;
	      #xSaveRecipe := FALSE;
	      #suiStepSaveRecipe := #stepCtrlRecipeNumber;
	      #sxRecipeSaved := FALSE;
	      
	    ELSIF #xDeleteRecipe THEN // User press delete recipe
	      #sxOperationInProgress := TRUE;
	      #xDeleteRecipe := FALSE;
	      #CurrentRecipe := #RecipeEmpty;
	      #WorkRecipe.RecipeName := #CurrentRecipe.RecipeName;
	      #WorkRecipe.RecipeCbsType := #CurrentRecipe.RecipeCbsType;
	      #WorkRecipe.RecipeRawMaterial := #CurrentRecipe.RecipeRawMaterial;
	      #WorkRecipe.RecipeTrajNumber := #CurrentRecipe.RecipeTrajNumber;
	      #WorkRecipe.RecipeLayerType.JobTableLeft[0] := #RecipeEmpty.RecipeLayerType[1].JobTableLeft[0];
	      #WorkRecipe.RecipeLayerType.JobTableRight[0] := #RecipeEmpty.RecipeLayerType[1].JobTableRight[0];
	      #usiJobNumberLeft := 0;
	      #usiJobNumberRight := 0;
	      #usiProcessPhase := 0;
	      #suiStepSaveRecipe := #stepCtrlRecipeNumber;
	      #sxRecipeSaved := FALSE;
	      
	    ELSIF #xUnloadRecipe THEN
	      #sxOperationInProgress := TRUE;
	      #xUnloadRecipe := FALSE;
	      #usiNumRecipe := 0;
	      #CurrentRecipe := #RecipeEmpty;
	      #WorkRecipe.RecipeName := #CurrentRecipe.RecipeName;
	      #WorkRecipe.RecipeCbsType := #CurrentRecipe.RecipeCbsType;
	      #WorkRecipe.RecipeRawMaterial := #CurrentRecipe.RecipeRawMaterial;
	      #WorkRecipe.RecipeTrajNumber := #CurrentRecipe.RecipeTrajNumber;
	      #WorkRecipe.RecipeLayerType.JobTableLeft[0] := #RecipeEmpty.RecipeLayerType[1].JobTableLeft[0];
	      #WorkRecipe.RecipeLayerType.JobTableRight[0] := #RecipeEmpty.RecipeLayerType[1].JobTableRight[0];
	      #usiJobNumberLeft := 0;
	      #usiJobNumberRight := 0;
	      #usiProcessPhase := 0;
	      #sxUpdateDisplayList := TRUE;
	      
	    END_IF;
	  END_REGION
	  
	END_IF;
	
	REGION Manage list of recipe on HMI
	  IF #suiIndexDisplay = 0 THEN // Initialization of display index
	    #suiIndexDisplay := 1;
	    #sxUpdateDisplayList := TRUE;
	  ELSIF #xNextRecipe THEN // User press next recipe
	    #xNextRecipe := FALSE;
	    IF #suiIndexDisplay <= 241 THEN
	      #suiIndexDisplay += 10;
	      #sxUpdateDisplayList := TRUE;
	    END_IF;
	  ELSIF #xPrevRecipe THEN // User pres previous recipe
	    #xPrevRecipe := FALSE;
	    IF #suiIndexDisplay >= 11 THEN
	      #suiIndexDisplay -= 10;
	      #sxUpdateDisplayList := TRUE;
	    END_IF;
	  END_IF;
	  
	  //IF #sxUpdateDisplayList THEN
	    //#sxUpdateDisplayList := FALSE;
	    IF ((#suiIndexDisplay > #suiTotalOfRecipe) AND (#suiIndexDisplay >= 11)) THEN
	      #suiIndexDisplay -= 10;
	      #sxUpdateDisplayList := TRUE;
	    END_IF;
	    FOR #suiCount_1 := 1 TO 10 DO
	      #aRecipeList[#suiCount_1].RecipeIndex := #aListRecipe[#suiIndexDisplay + (#suiCount_1 - 1)].RecipeIndex;
	      #aRecipeList[#suiCount_1].RecipeName := #aListRecipe[#suiIndexDisplay + (#suiCount_1 - 1)].RecipeName;
	      #aRecipeList[#suiCount_1].RecipeSelected := (#aRecipeList[#suiCount_1].RecipeIndex = #usiNumRecipe) AND (#usiNumRecipe <> 0);
	      IF #sxOperationInProgress OR #xSandingInProgress THEN
	        #aRecipeList[#suiCount_1].RecipeIndex := 0;
	      END_IF;
	    END_FOR;
	  //END_IF;
	  
	  
	END_REGION
	
	REGION Processing phase change
	  
	  IF ((#usiProcessPhase <> #susiMemProcessPhase) AND (#usiProcessPhase <> 0)) THEN
	    #susiMemProcessPhase := #usiProcessPhase;
	    #usiJobNumberLeft := 0;
	    #usiJobNumberRight := 0;
	    #WorkRecipe.RecipeLayerType := #CurrentRecipe.RecipeLayerType[#usiProcessPhase];
	    #WorkRecipe.RecipeLayerType.JobTableLeft[0] := #RecipeEmpty.RecipeLayerType[1].JobTableLeft[0];
	    #WorkRecipe.RecipeLayerType.JobTableRight[0] := #RecipeEmpty.RecipeLayerType[1].JobTableRight[0];
	  ELSIF ((#usiProcessPhase <> #susiMemProcessPhase) AND (#usiProcessPhase = 0)) THEN
	    #susiMemProcessPhase := 0;
	    #usiJobNumberLeft := 0;
	    #usiJobNumberRight := 0;
	    #WorkRecipe.RecipeLayerType := #RecipeEmpty.RecipeLayerType[1];
	    #WorkRecipe.RecipeLayerType.JobTableLeft[0] := #RecipeEmpty.RecipeLayerType[1].JobTableLeft[0];
	    #WorkRecipe.RecipeLayerType.JobTableRight[0] := #RecipeEmpty.RecipeLayerType[1].JobTableRight[0];
	  END_IF;
	  
	END_REGION
	
	REGION Manage Button on HMI
	  // Display or hide Next button
	  #xDisplayNextButton := ((#suiIndexDisplay + 9) < #suiTotalOfRecipe);
	  // Display or hide Previous button
	  #xDisplayPrevButton := (#suiIndexDisplay > 10);
	  // Diseable or enable Delte recipe button
	  #xDiseableDeleteButton := #sxOperationInProgress OR #xSandingInProgress OR (#usiNumRecipe = 0);
	  // Diseable or enable New recipe button
	  #xDiseableNewButton := #sxOperationInProgress OR #xSandingInProgress;
	  // Diseable or enable Save recipe button
	  #xDiseableSaveButton := #sxOperationInProgress OR (#usiNumRecipe = 0);
	  // Lock or unlock the modification of the recipe
	  #xLockRecipe := (#usiNumRecipe = 0) (*OR (#usiProcessPhase = 0)*) OR #xSandingInProgress;
	  // Lock or unlock selection of job data number
	  #xLockSelectJobDataNumber := (#usiNumRecipe = 0) OR (#usiProcessPhase = 0);
	  // Lock or unlock modification of job data Left Robot
	  #xLockJobDataLeft := (#usiNumRecipe = 0) OR (#usiProcessPhase = 0) OR (#usiJobNumberLeft = 0);
	  // Lock or unlock modification of job data Right Robot
	  #xLockJobDataRight := (#usiNumRecipe = 0) OR (#usiProcessPhase = 0) OR (#usiJobNumberRight = 0);
	  
	  #miDB_FPLockSelectRecipe(CLK:=(#sxOperationInProgress OR #xSandingInProgress));
	  #miDB_FNLockSelectRecipe(CLK:=(NOT #sxOperationInProgress) AND (NOT #xSandingInProgress));
	  
	  IF #miDB_FPLockSelectRecipe.Q OR #miDB_FNLockSelectRecipe.Q THEN
	    #sxUpdateDisplayList := TRUE;
	 END_IF;
	 
	END_REGION
	
	REGION Function
	  // Read only one recipe in the data base
	  #txReqReadRecipe := (#suiStepLoadRecipe = #stepStartLoadRecipe);
	  #snReadDblResult := READ_DBL(REQ := #txReqReadRecipe, SRCBLK := #aRecipesDB[#usiNumRecipe], BUSY => #sxReadDblBusy, DSTBLK => #CurrentRecipe);
	  
	  // Read all the recipe in the data base
	  #txReqListRecipe := (#suiStepListRecipe = #stepStartListLoadRecipe);
	  #snListDblResult := READ_DBL(REQ := #txReqListRecipe, SRCBLK := #aRecipesDB[#susiCurrentIndexList], BUSY => #sxListDblBusy, DSTBLK => #TempRecipe);
	  
	  // Write the current recipe in the data base
	  #txReqWriteRecipe := (#suiStepSaveRecipe = #stepStartSaveRecipe);
	  #snWriteDblResult := WRIT_DBL(REQ := #txReqWriteRecipe, SRCBLK := #CurrentRecipe, BUSY => #sxWriteDblBusy, DSTBLK => #aRecipesDB[#usiNumRecipe]);
	END_REGION
	
	
	
END_FUNCTION_BLOCK

FUNCTION "FC60_Fault" : Void   // FC60, LAD
{ S7_Optimized_Access := 'TRUE' }
// stored: AutoNumber false, IsIECCheckEnabled true, SetENOAutomatically false
   VAR_TEMP
      txFaultMaster : Bool;
      txFaultLeft : Bool;
      txFaultRight : Bool;
   END_VAR
BEGIN

REGION Network 1: Safety fault
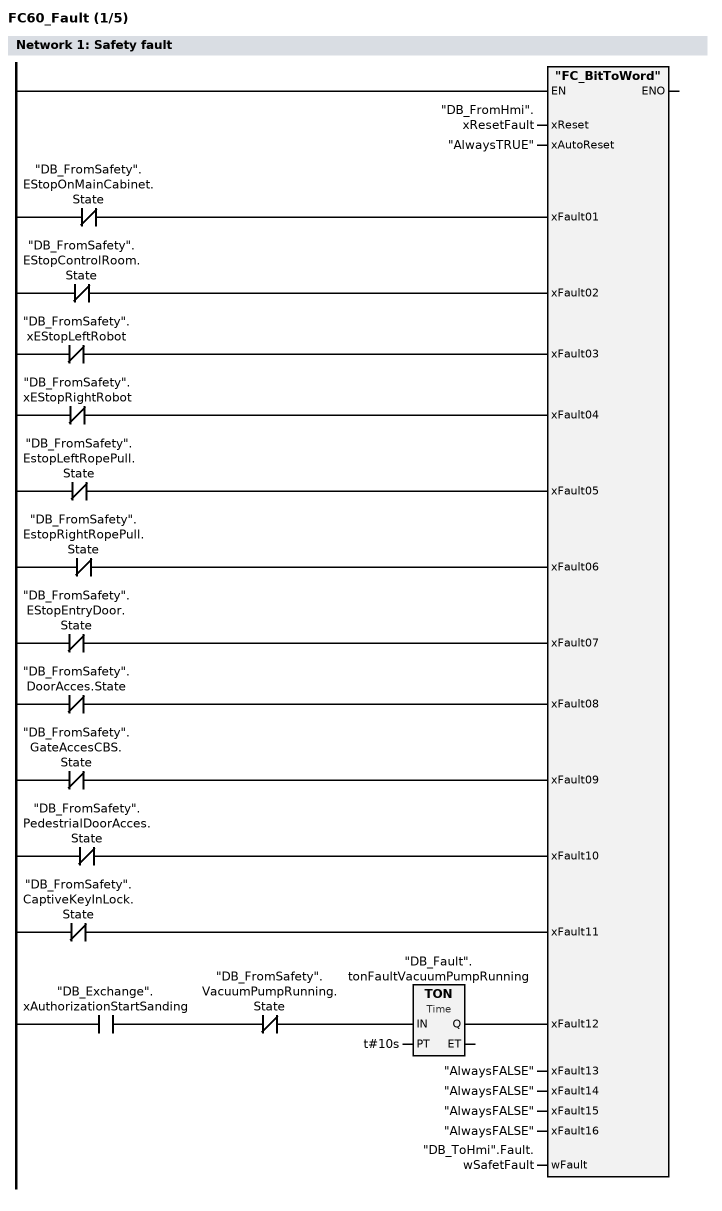
   RUNG wire#powerrail
      "FC_BitToWord"(xFault01 := wire#w1, xFault02 := wire#w2, xFault03 := wire#w3, xFault04 := wire#w4, xFault05 := wire#w5, xFault06 := wire#w6, xFault07 := wire#w7, xFault08 := wire#w8, xFault09 := wire#w9, xFault10 := wire#w10, xFault11 := wire#w11, xFault12 := wire#w12, xReset := "DB_FromHmi".xResetFault, xAutoReset := "AlwaysTRUE", xFault13 := "AlwaysFALSE", xFault14 := "AlwaysFALSE", xFault15 := "AlwaysFALSE", xFault16 := "AlwaysFALSE", wFault := "DB_ToHmi".Fault.wSafetFault)
   END_RUNG
   RUNG wire#powerrail
      I_Contact( "DB_FromSafety".EStopOnMainCabinet.State )
   END_RUNG wire#w1
   RUNG wire#powerrail
      I_Contact( "DB_FromSafety".EStopControlRoom.State )
   END_RUNG wire#w2
   RUNG wire#powerrail
      I_Contact( "DB_FromSafety".xEStopLeftRobot )
   END_RUNG wire#w3
   RUNG wire#powerrail
      I_Contact( "DB_FromSafety".xEStopRightRobot )
   END_RUNG wire#w4
   RUNG wire#powerrail
      I_Contact( "DB_FromSafety".EstopLeftRopePull.State )
   END_RUNG wire#w5
   RUNG wire#powerrail
      I_Contact( "DB_FromSafety".EstopRightRopePull.State )
   END_RUNG wire#w6
   RUNG wire#powerrail
      I_Contact( "DB_FromSafety".EStopEntryDoor.State )
   END_RUNG wire#w7
   RUNG wire#powerrail
      I_Contact( "DB_FromSafety".DoorAcces.State )
   END_RUNG wire#w8
   RUNG wire#powerrail
      I_Contact( "DB_FromSafety".GateAccesCBS.State )
   END_RUNG wire#w9
   RUNG wire#powerrail
      I_Contact( "DB_FromSafety".PedestrialDoorAcces.State )
   END_RUNG wire#w10
   RUNG wire#powerrail
      I_Contact( "DB_FromSafety".CaptiveKeyInLock.State )
   END_RUNG wire#w11
   RUNG wire#powerrail
      Contact( "DB_Exchange".xAuthorizationStartSanding )
      I_Contact( "DB_FromSafety".VacuumPumpRunning.State )
      { S7_Templates := "time_type := Time" } "DB_Fault".tonFaultVacuumPumpRunning.TON(pt := t#10s, et =>)
   END_RUNG wire#w12
   // the same network as SCL:
   "DB_Fault".tonFaultVacuumPumpRunning.TON(IN := "DB_Exchange".xAuthorizationStartSanding AND NOT "DB_FromSafety".VacuumPumpRunning.State,
                           PT := t#10s);
   "FC_BitToWord"(xReset := "DB_FromHmi".xResetFault,
                  xAutoReset := "AlwaysTRUE",
                  xFault01 := NOT "DB_FromSafety".EStopOnMainCabinet.State,
                  xFault02 := NOT "DB_FromSafety".EStopControlRoom.State,
                  xFault03 := NOT "DB_FromSafety".xEStopLeftRobot,
                  xFault04 := NOT "DB_FromSafety".xEStopRightRobot,
                  xFault05 := NOT "DB_FromSafety".EstopLeftRopePull.State,
                  xFault06 := NOT "DB_FromSafety".EstopRightRopePull.State,
                  xFault07 := NOT "DB_FromSafety".EStopEntryDoor.State,
                  xFault08 := NOT "DB_FromSafety".DoorAcces.State,
                  xFault09 := NOT "DB_FromSafety".GateAccesCBS.State,
                  xFault10 := NOT "DB_FromSafety".PedestrialDoorAcces.State,
                  xFault11 := NOT "DB_FromSafety".CaptiveKeyInLock.State,
                  xFault12 := "DB_Fault".tonFaultVacuumPumpRunning.Q,
                  xFault13 := "AlwaysFALSE",
                  xFault14 := "AlwaysFALSE",
                  xFault15 := "AlwaysFALSE",
                  xFault16 := "AlwaysFALSE",
                  wFault := "DB_ToHmi".Fault.wSafetFault);
END_REGION

REGION Network 2: Error safety module
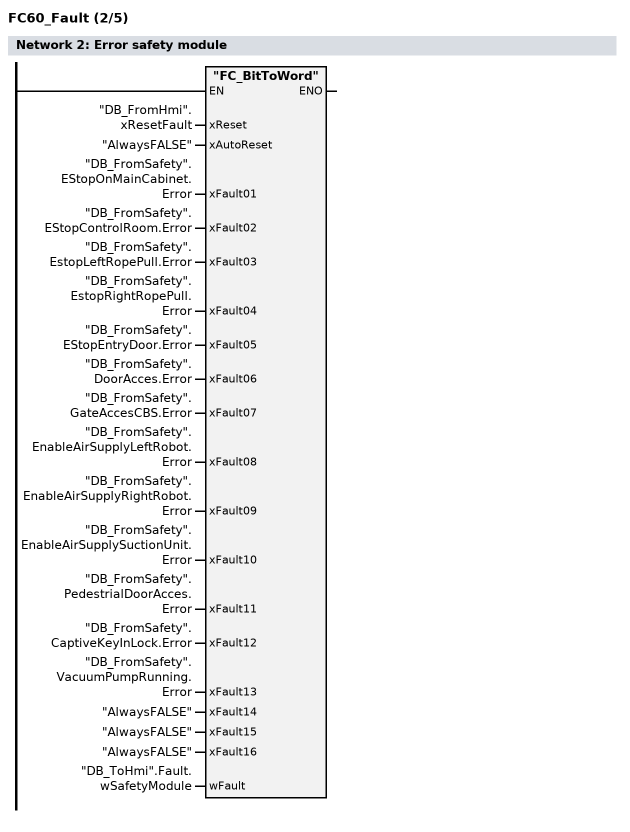
   RUNG wire#powerrail
      "FC_BitToWord"(xReset := "DB_FromHmi".xResetFault, xAutoReset := "AlwaysFALSE", xFault01 := "DB_FromSafety".EStopOnMainCabinet.Error, xFault02 := "DB_FromSafety".EStopControlRoom.Error, xFault03 := "DB_FromSafety".EstopLeftRopePull.Error, xFault04 := "DB_FromSafety".EstopRightRopePull.Error, xFault05 := "DB_FromSafety".EStopEntryDoor.Error, xFault06 := "DB_FromSafety".DoorAcces.Error, xFault07 := "DB_FromSafety".GateAccesCBS.Error, xFault08 := "DB_FromSafety".EnableAirSupplyLeftRobot.Error, xFault09 := "DB_FromSafety".EnableAirSupplyRightRobot.Error, xFault10 := "DB_FromSafety".EnableAirSupplySuctionUnit.Error, xFault11 := "DB_FromSafety".PedestrialDoorAcces.Error, xFault12 := "DB_FromSafety".CaptiveKeyInLock.Error, xFault13 := "DB_FromSafety".VacuumPumpRunning.Error, xFault14 := "AlwaysFALSE", xFault15 := "AlwaysFALSE", xFault16 := "AlwaysFALSE", wFault := "DB_ToHmi".Fault.wSafetyModule)
   END_RUNG
   // the same network as SCL:
   "FC_BitToWord"(xReset := "DB_FromHmi".xResetFault,
                  xAutoReset := "AlwaysFALSE",
                  xFault01 := "DB_FromSafety".EStopOnMainCabinet.Error,
                  xFault02 := "DB_FromSafety".EStopControlRoom.Error,
                  xFault03 := "DB_FromSafety".EstopLeftRopePull.Error,
                  xFault04 := "DB_FromSafety".EstopRightRopePull.Error,
                  xFault05 := "DB_FromSafety".EStopEntryDoor.Error,
                  xFault06 := "DB_FromSafety".DoorAcces.Error,
                  xFault07 := "DB_FromSafety".GateAccesCBS.Error,
                  xFault08 := "DB_FromSafety".EnableAirSupplyLeftRobot.Error,
                  xFault09 := "DB_FromSafety".EnableAirSupplyRightRobot.Error,
                  xFault10 := "DB_FromSafety".EnableAirSupplySuctionUnit.Error,
                  xFault11 := "DB_FromSafety".PedestrialDoorAcces.Error,
                  xFault12 := "DB_FromSafety".CaptiveKeyInLock.Error,
                  xFault13 := "DB_FromSafety".VacuumPumpRunning.Error,
                  xFault14 := "AlwaysFALSE",
                  xFault15 := "AlwaysFALSE",
                  xFault16 := "AlwaysFALSE",
                  wFault := "DB_ToHmi".Fault.wSafetyModule);
END_REGION

REGION Network 3: Other fault on Master PLC
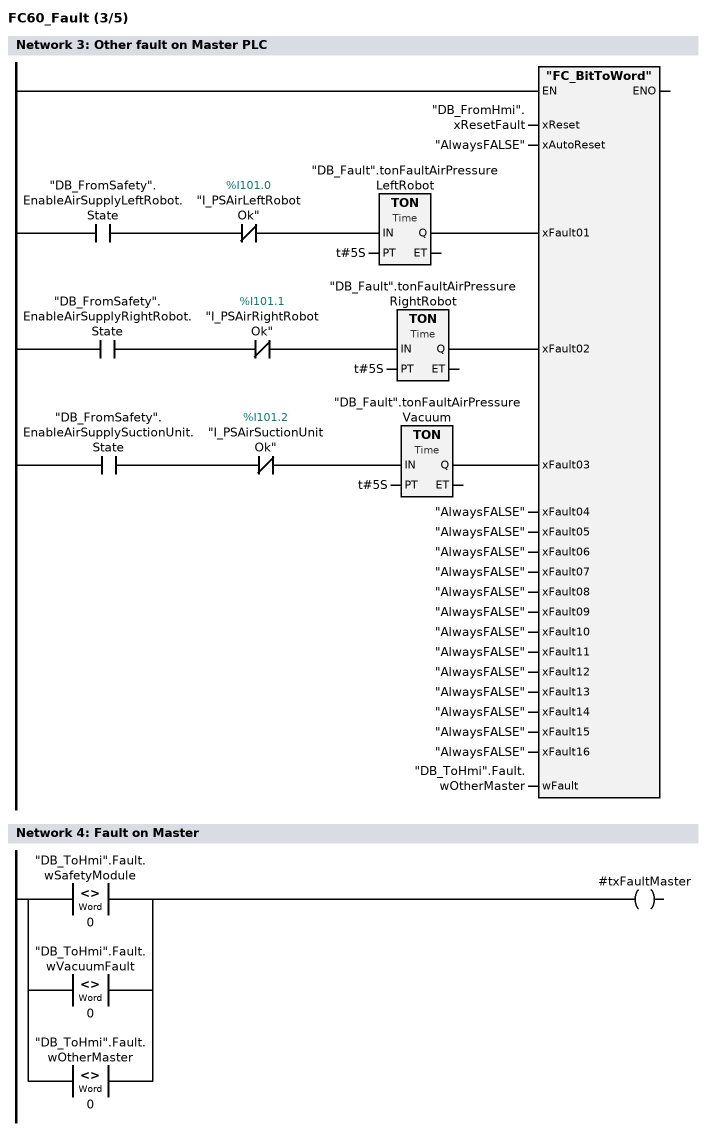
   RUNG wire#powerrail
      "FC_BitToWord"(xFault01 := wire#w1, xFault02 := wire#w2, xFault03 := wire#w3, xReset := "DB_FromHmi".xResetFault, xAutoReset := "AlwaysFALSE", xFault04 := "AlwaysFALSE", xFault05 := "AlwaysFALSE", xFault06 := "AlwaysFALSE", xFault07 := "AlwaysFALSE", xFault08 := "AlwaysFALSE", xFault09 := "AlwaysFALSE", xFault10 := "AlwaysFALSE", xFault11 := "AlwaysFALSE", xFault12 := "AlwaysFALSE", xFault13 := "AlwaysFALSE", xFault14 := "AlwaysFALSE", xFault15 := "AlwaysFALSE", xFault16 := "AlwaysFALSE", wFault := "DB_ToHmi".Fault.wOtherMaster)
   END_RUNG
   RUNG wire#powerrail
      Contact( "DB_FromSafety".EnableAirSupplyLeftRobot.State )
      I_Contact( "I_PSAirLeftRobotOk" )
      { S7_Templates := "time_type := Time" } "DB_Fault".tonFaultAirPressureLeftRobot.TON(pt := t#5S, et =>)
   END_RUNG wire#w1
   RUNG wire#powerrail
      Contact( "DB_FromSafety".EnableAirSupplyRightRobot.State )
      I_Contact( "I_PSAirRightRobotOk" )
      { S7_Templates := "time_type := Time" } "DB_Fault".tonFaultAirPressureRightRobot.TON(pt := t#5S, et =>)
   END_RUNG wire#w2
   RUNG wire#powerrail
      Contact( "DB_FromSafety".EnableAirSupplySuctionUnit.State )
      I_Contact( "I_PSAirSuctionUnitOk" )
      { S7_Templates := "time_type := Time" } "DB_Fault".tonFaultAirPressureVacuum.TON(pt := t#5S, et =>)
   END_RUNG wire#w3
   // the same network as SCL:
   "DB_Fault".tonFaultAirPressureLeftRobot.TON(IN := "DB_FromSafety".EnableAirSupplyLeftRobot.State AND NOT "I_PSAirLeftRobotOk",
                           PT := t#5S);
   "DB_Fault".tonFaultAirPressureRightRobot.TON(IN := "DB_FromSafety".EnableAirSupplyRightRobot.State AND NOT "I_PSAirRightRobotOk",
                           PT := t#5S);
   "DB_Fault".tonFaultAirPressureVacuum.TON(IN := "DB_FromSafety".EnableAirSupplySuctionUnit.State AND NOT "I_PSAirSuctionUnitOk",
                           PT := t#5S);
   "FC_BitToWord"(xReset := "DB_FromHmi".xResetFault,
                  xAutoReset := "AlwaysFALSE",
                  xFault01 := "DB_Fault".tonFaultAirPressureLeftRobot.Q,
                  xFault02 := "DB_Fault".tonFaultAirPressureRightRobot.Q,
                  xFault03 := "DB_Fault".tonFaultAirPressureVacuum.Q,
                  xFault04 := "AlwaysFALSE",
                  xFault05 := "AlwaysFALSE",
                  xFault06 := "AlwaysFALSE",
                  xFault07 := "AlwaysFALSE",
                  xFault08 := "AlwaysFALSE",
                  xFault09 := "AlwaysFALSE",
                  xFault10 := "AlwaysFALSE",
                  xFault11 := "AlwaysFALSE",
                  xFault12 := "AlwaysFALSE",
                  xFault13 := "AlwaysFALSE",
                  xFault14 := "AlwaysFALSE",
                  xFault15 := "AlwaysFALSE",
                  xFault16 := "AlwaysFALSE",
                  wFault := "DB_ToHmi".Fault.wOtherMaster);
END_REGION

REGION Network 4: Fault on Master
   RUNG wire#powerrail
      { S7_Templates := "SrcType := Word" } NE_Contact(in1 := "DB_ToHmi".Fault.wSafetyModule, in2 := 0)
      wire#w1
      Coil( #txFaultMaster )
   END_RUNG
   RUNG wire#powerrail
      { S7_Templates := "SrcType := Word" } NE_Contact(in1 := "DB_ToHmi".Fault.wVacuumFault, in2 := 0)
   END_RUNG wire#w1
   RUNG wire#powerrail
      { S7_Templates := "SrcType := Word" } NE_Contact(in1 := "DB_ToHmi".Fault.wOtherMaster, in2 := 0)
   END_RUNG wire#w1
   // the same network as SCL:
   #txFaultMaster := ("DB_ToHmi".Fault.wSafetyModule <> 0) OR ("DB_ToHmi".Fault.wVacuumFault <> 0) OR ("DB_ToHmi".Fault.wOtherMaster <> 0);
END_REGION

REGION Network 5: Fault on Left
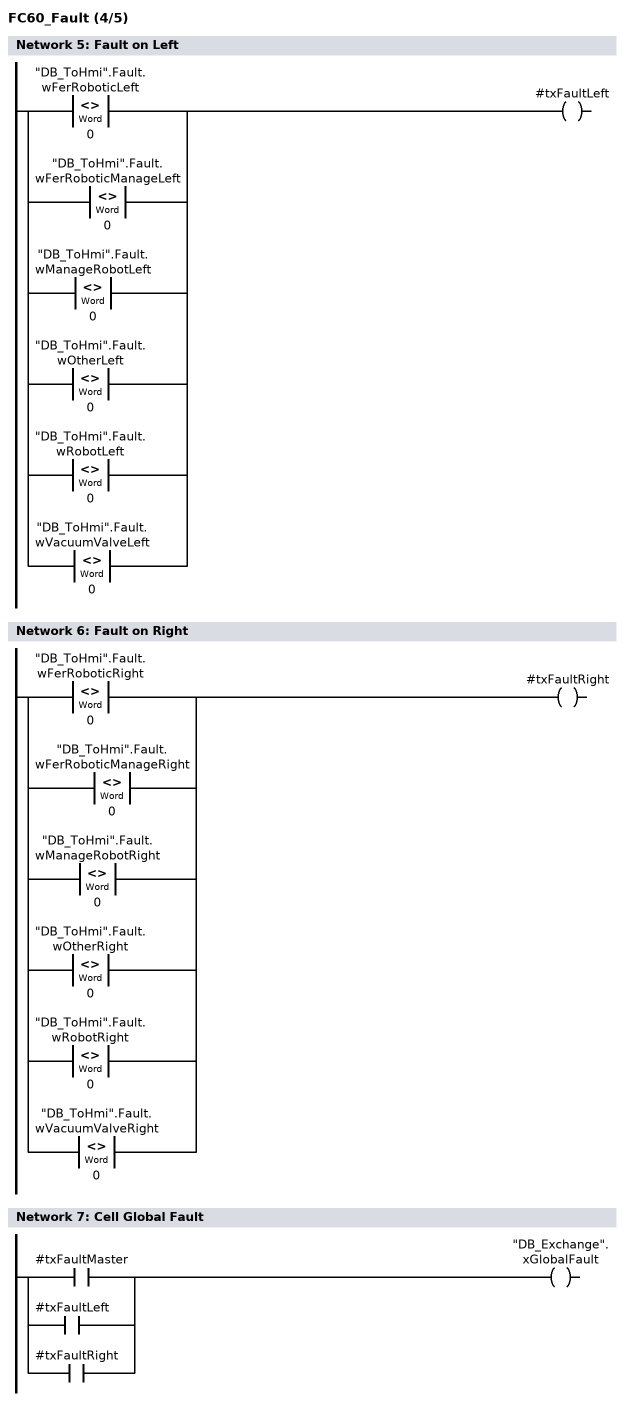
   RUNG wire#powerrail
      { S7_Templates := "SrcType := Word" } NE_Contact(in1 := "DB_ToHmi".Fault.wFerRoboticLeft, in2 := 0)
      wire#w1
      Coil( #txFaultLeft )
   END_RUNG
   RUNG wire#powerrail
      { S7_Templates := "SrcType := Word" } NE_Contact(in1 := "DB_ToHmi".Fault.wFerRoboticManageLeft, in2 := 0)
   END_RUNG wire#w1
   RUNG wire#powerrail
      { S7_Templates := "SrcType := Word" } NE_Contact(in1 := "DB_ToHmi".Fault.wManageRobotLeft, in2 := 0)
   END_RUNG wire#w1
   RUNG wire#powerrail
      { S7_Templates := "SrcType := Word" } NE_Contact(in1 := "DB_ToHmi".Fault.wOtherLeft, in2 := 0)
   END_RUNG wire#w1
   RUNG wire#powerrail
      { S7_Templates := "SrcType := Word" } NE_Contact(in1 := "DB_ToHmi".Fault.wRobotLeft, in2 := 0)
   END_RUNG wire#w1
   RUNG wire#powerrail
      { S7_Templates := "SrcType := Word" } NE_Contact(in1 := "DB_ToHmi".Fault.wVacuumValveLeft, in2 := 0)
   END_RUNG wire#w1
   // the same network as SCL:
   #txFaultLeft := ("DB_ToHmi".Fault.wFerRoboticLeft <> 0) OR ("DB_ToHmi".Fault.wFerRoboticManageLeft <> 0) OR ("DB_ToHmi".Fault.wManageRobotLeft <> 0) OR ("DB_ToHmi".Fault.wOtherLeft <> 0) OR ("DB_ToHmi".Fault.wRobotLeft <> 0) OR ("DB_ToHmi".Fault.wVacuumValveLeft <> 0);
END_REGION

REGION Network 6: Fault on Right
   RUNG wire#powerrail
      { S7_Templates := "SrcType := Word" } NE_Contact(in1 := "DB_ToHmi".Fault.wFerRoboticRight, in2 := 0)
      wire#w1
      Coil( #txFaultRight )
   END_RUNG
   RUNG wire#powerrail
      { S7_Templates := "SrcType := Word" } NE_Contact(in1 := "DB_ToHmi".Fault.wFerRoboticManageRight, in2 := 0)
   END_RUNG wire#w1
   RUNG wire#powerrail
      { S7_Templates := "SrcType := Word" } NE_Contact(in1 := "DB_ToHmi".Fault.wManageRobotRight, in2 := 0)
   END_RUNG wire#w1
   RUNG wire#powerrail
      { S7_Templates := "SrcType := Word" } NE_Contact(in1 := "DB_ToHmi".Fault.wOtherRight, in2 := 0)
   END_RUNG wire#w1
   RUNG wire#powerrail
      { S7_Templates := "SrcType := Word" } NE_Contact(in1 := "DB_ToHmi".Fault.wRobotRight, in2 := 0)
   END_RUNG wire#w1
   RUNG wire#powerrail
      { S7_Templates := "SrcType := Word" } NE_Contact(in1 := "DB_ToHmi".Fault.wVacuumValveRight, in2 := 0)
   END_RUNG wire#w1
   // the same network as SCL:
   #txFaultRight := ("DB_ToHmi".Fault.wFerRoboticRight <> 0) OR ("DB_ToHmi".Fault.wFerRoboticManageRight <> 0) OR ("DB_ToHmi".Fault.wManageRobotRight <> 0) OR ("DB_ToHmi".Fault.wOtherRight <> 0) OR ("DB_ToHmi".Fault.wRobotRight <> 0) OR ("DB_ToHmi".Fault.wVacuumValveRight <> 0);
END_REGION

REGION Network 7: Cell Global Fault
   RUNG wire#powerrail
      Contact( #txFaultMaster )
      wire#w1
      Coil( "DB_Exchange".xGlobalFault )
   END_RUNG
   RUNG wire#powerrail
      Contact( #txFaultLeft )
   END_RUNG wire#w1
   RUNG wire#powerrail
      Contact( #txFaultRight )
   END_RUNG wire#w1
   // the same network as SCL:
   "DB_Exchange".xGlobalFault := #txFaultMaster OR #txFaultLeft OR #txFaultRight;
END_REGION

REGION Network 8: Cell Global warning
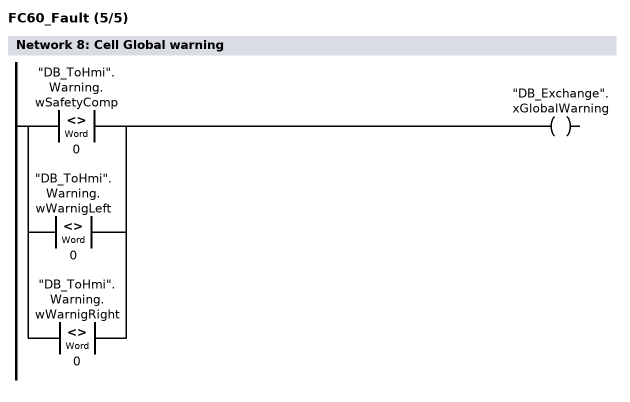
   RUNG wire#powerrail
      { S7_Templates := "SrcType := Word" } NE_Contact(in1 := "DB_ToHmi".Warning.wSafetyComp, in2 := 0)
      wire#w1
      Coil( "DB_Exchange".xGlobalWarning )
   END_RUNG
   RUNG wire#powerrail
      { S7_Templates := "SrcType := Word" } NE_Contact(in1 := "DB_ToHmi".Warning.wWarnigLeft, in2 := 0)
   END_RUNG wire#w1
   RUNG wire#powerrail
      { S7_Templates := "SrcType := Word" } NE_Contact(in1 := "DB_ToHmi".Warning.wWarnigRight, in2 := 0)
   END_RUNG wire#w1
   // the same network as SCL:
   "DB_Exchange".xGlobalWarning := ("DB_ToHmi".Warning.wSafetyComp <> 0) OR ("DB_ToHmi".Warning.wWarnigLeft <> 0) OR ("DB_ToHmi".Warning.wWarnigRight <> 0);
END_REGION
END_FUNCTION

FUNCTION "FC70_RecordData" : Void   // FC70, LAD
{ S7_Optimized_Access := 'TRUE' }
// stored: AutoNumber false, SetENOAutomatically false
   VAR_TEMP   // added for the SCL form of the ladder/FBD networks
      _w1 : Bool;
   END_VAR
BEGIN

REGION Network 1: Record Production data
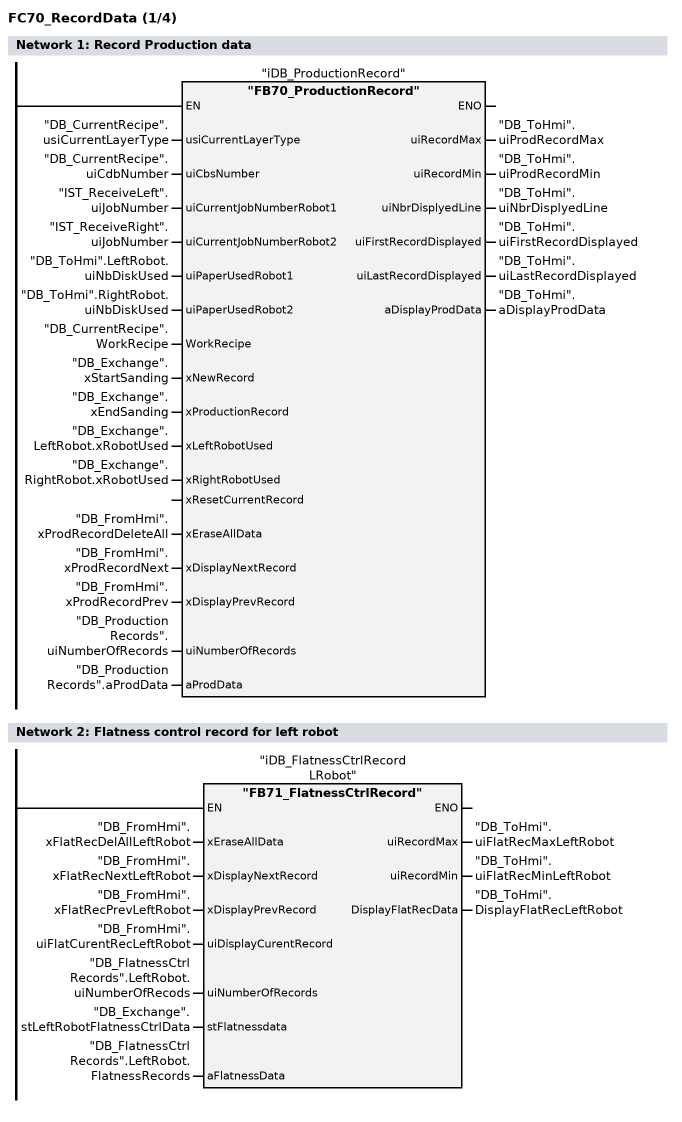
   RUNG wire#powerrail
      "iDB_ProductionRecord"(usiCurrentLayerType := "DB_CurrentRecipe".usiCurrentLayerType, uiCbsNumber := "DB_CurrentRecipe".uiCdbNumber, uiCurrentJobNumberRobot1 := "IST_ReceiveLeft".uiJobNumber, uiCurrentJobNumberRobot2 := "IST_ReceiveRight".uiJobNumber, uiPaperUsedRobot1 := "DB_ToHmi".LeftRobot.uiNbDiskUsed, uiPaperUsedRobot2 := "DB_ToHmi".RightRobot.uiNbDiskUsed, WorkRecipe := "DB_CurrentRecipe".WorkRecipe, xNewRecord := "DB_Exchange".xStartSanding, xProductionRecord := "DB_Exchange".xEndSanding, xLeftRobotUsed := "DB_Exchange".LeftRobot.xRobotUsed, xRightRobotUsed := "DB_Exchange".RightRobot.xRobotUsed, xResetCurrentRecord :=, xEraseAllData := "DB_FromHmi".xProdRecordDeleteAll, xDisplayNextRecord := "DB_FromHmi".xProdRecordNext, xDisplayPrevRecord := "DB_FromHmi".xProdRecordPrev, uiNumberOfRecords := "DB_ProductionRecords".uiNumberOfRecords, aProdData := "DB_ProductionRecords".aProdData, uiRecordMax => "DB_ToHmi".uiProdRecordMax, uiRecordMin => "DB_ToHmi".uiProdRecordMin, uiNbrDisplyedLine => "DB_ToHmi".uiNbrDisplyedLine, uiFirstRecordDisplayed => "DB_ToHmi".uiFirstRecordDisplayed, uiLastRecordDisplayed => "DB_ToHmi".uiLastRecordDisplayed, aDisplayProdData => "DB_ToHmi".aDisplayProdData)
   END_RUNG
   // the same network as SCL:
   "iDB_ProductionRecord"(usiCurrentLayerType := "DB_CurrentRecipe".usiCurrentLayerType,   // "FB70_ProductionRecord"
                          uiCbsNumber := "DB_CurrentRecipe".uiCdbNumber,
                          uiCurrentJobNumberRobot1 := "IST_ReceiveLeft".uiJobNumber,
                          uiCurrentJobNumberRobot2 := "IST_ReceiveRight".uiJobNumber,
                          uiPaperUsedRobot1 := "DB_ToHmi".LeftRobot.uiNbDiskUsed,
                          uiPaperUsedRobot2 := "DB_ToHmi".RightRobot.uiNbDiskUsed,
                          WorkRecipe := "DB_CurrentRecipe".WorkRecipe,
                          xNewRecord := "DB_Exchange".xStartSanding,
                          xProductionRecord := "DB_Exchange".xEndSanding,
                          xLeftRobotUsed := "DB_Exchange".LeftRobot.xRobotUsed,
                          xRightRobotUsed := "DB_Exchange".RightRobot.xRobotUsed,
                          xEraseAllData := "DB_FromHmi".xProdRecordDeleteAll,
                          xDisplayNextRecord := "DB_FromHmi".xProdRecordNext,
                          xDisplayPrevRecord := "DB_FromHmi".xProdRecordPrev,
                          uiNumberOfRecords := "DB_ProductionRecords".uiNumberOfRecords,
                          aProdData := "DB_ProductionRecords".aProdData,
                          uiRecordMax => "DB_ToHmi".uiProdRecordMax,
                          uiRecordMin => "DB_ToHmi".uiProdRecordMin,
                          uiNbrDisplyedLine => "DB_ToHmi".uiNbrDisplyedLine,
                          uiFirstRecordDisplayed => "DB_ToHmi".uiFirstRecordDisplayed,
                          uiLastRecordDisplayed => "DB_ToHmi".uiLastRecordDisplayed,
                          aDisplayProdData => "DB_ToHmi".aDisplayProdData);
END_REGION

REGION Network 2: Flatness control record for left robot
   RUNG wire#powerrail
      "iDB_FlatnessCtrlRecordLRobot"(xEraseAllData := "DB_FromHmi".xFlatRecDelAllLeftRobot, xDisplayNextRecord := "DB_FromHmi".xFlatRecNextLeftRobot, xDisplayPrevRecord := "DB_FromHmi".xFlatRecPrevLeftRobot, uiDisplayCurentRecord := "DB_FromHmi".uiFlatCurentRecLeftRobot, uiNumberOfRecords := "DB_FlatnessCtrlRecords".LeftRobot.uiNumberOfRecods, stFlatnessdata := "DB_Exchange".stLeftRobotFlatnessCtrlData, aFlatnessData := "DB_FlatnessCtrlRecords".LeftRobot.FlatnessRecords, uiRecordMax => "DB_ToHmi".uiFlatRecMaxLeftRobot, uiRecordMin => "DB_ToHmi".uiFlatRecMinLeftRobot, DisplayFlatRecData => "DB_ToHmi".DisplayFlatRecLeftRobot)
   END_RUNG
   // the same network as SCL:
   "iDB_FlatnessCtrlRecordLRobot"(xEraseAllData := "DB_FromHmi".xFlatRecDelAllLeftRobot,   // "FB71_FlatnessCtrlRecord"
                           xDisplayNextRecord := "DB_FromHmi".xFlatRecNextLeftRobot,
                           xDisplayPrevRecord := "DB_FromHmi".xFlatRecPrevLeftRobot,
                           uiDisplayCurentRecord := "DB_FromHmi".uiFlatCurentRecLeftRobot,
                           uiNumberOfRecords := "DB_FlatnessCtrlRecords".LeftRobot.uiNumberOfRecods,
                           stFlatnessdata := "DB_Exchange".stLeftRobotFlatnessCtrlData,
                           aFlatnessData := "DB_FlatnessCtrlRecords".LeftRobot.FlatnessRecords,
                           uiRecordMax => "DB_ToHmi".uiFlatRecMaxLeftRobot,
                           uiRecordMin => "DB_ToHmi".uiFlatRecMinLeftRobot,
                           DisplayFlatRecData => "DB_ToHmi".DisplayFlatRecLeftRobot);
END_REGION

REGION Network 3: Flatness control record for Right robot
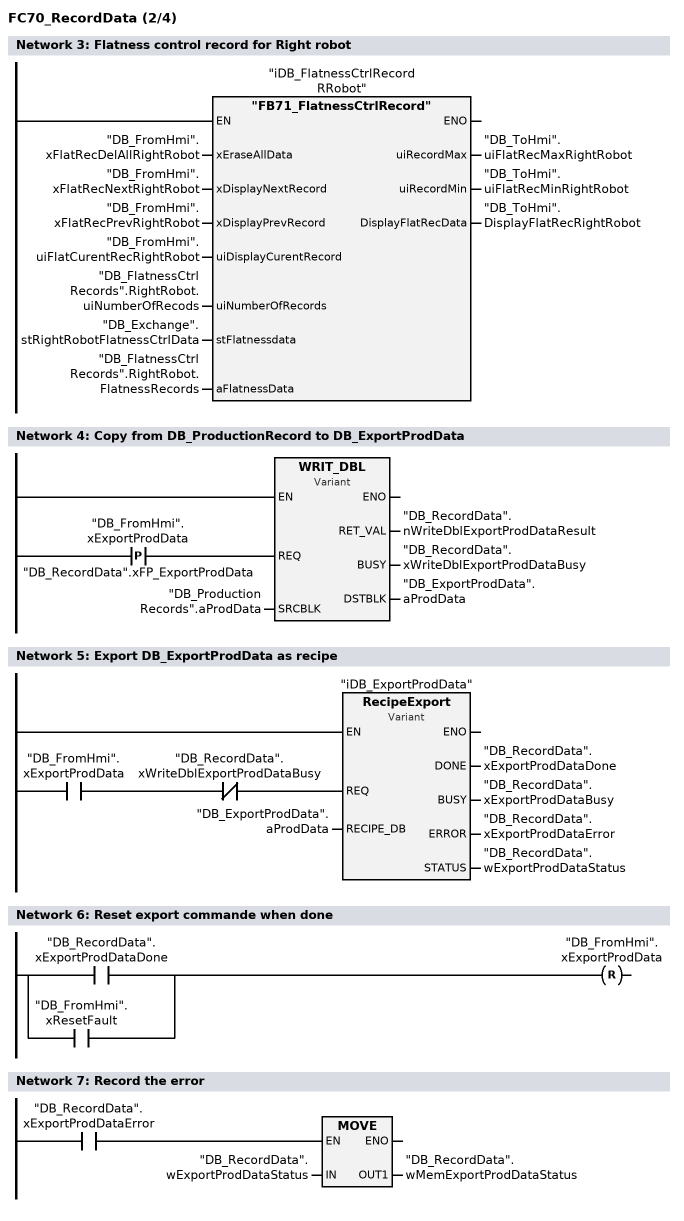
   RUNG wire#powerrail
      "iDB_FlatnessCtrlRecordRRobot"(xEraseAllData := "DB_FromHmi".xFlatRecDelAllRightRobot, xDisplayNextRecord := "DB_FromHmi".xFlatRecNextRightRobot, xDisplayPrevRecord := "DB_FromHmi".xFlatRecPrevRightRobot, uiDisplayCurentRecord := "DB_FromHmi".uiFlatCurentRecRightRobot, uiNumberOfRecords := "DB_FlatnessCtrlRecords".RightRobot.uiNumberOfRecods, stFlatnessdata := "DB_Exchange".stRightRobotFlatnessCtrlData, aFlatnessData := "DB_FlatnessCtrlRecords".RightRobot.FlatnessRecords, uiRecordMax => "DB_ToHmi".uiFlatRecMaxRightRobot, uiRecordMin => "DB_ToHmi".uiFlatRecMinRightRobot, DisplayFlatRecData => "DB_ToHmi".DisplayFlatRecRightRobot)
   END_RUNG
   // the same network as SCL:
   "iDB_FlatnessCtrlRecordRRobot"(xEraseAllData := "DB_FromHmi".xFlatRecDelAllRightRobot,   // "FB71_FlatnessCtrlRecord"
                           xDisplayNextRecord := "DB_FromHmi".xFlatRecNextRightRobot,
                           xDisplayPrevRecord := "DB_FromHmi".xFlatRecPrevRightRobot,
                           uiDisplayCurentRecord := "DB_FromHmi".uiFlatCurentRecRightRobot,
                           uiNumberOfRecords := "DB_FlatnessCtrlRecords".RightRobot.uiNumberOfRecods,
                           stFlatnessdata := "DB_Exchange".stRightRobotFlatnessCtrlData,
                           aFlatnessData := "DB_FlatnessCtrlRecords".RightRobot.FlatnessRecords,
                           uiRecordMax => "DB_ToHmi".uiFlatRecMaxRightRobot,
                           uiRecordMin => "DB_ToHmi".uiFlatRecMinRightRobot,
                           DisplayFlatRecData => "DB_ToHmi".DisplayFlatRecRightRobot);
END_REGION

REGION Network 4: Copy from DB_ProductionRecord to DB_ExportProdData
   RUNG wire#powerrail
      { S7_Templates := "[src_type := Variant, dest_type := Variant]" } WRIT_DBL(REQ := wire#w1, SRCBLK := "DB_ProductionRecords".aProdData, RET_VAL => "DB_RecordData".nWriteDblExportProdDataResult, BUSY => "DB_RecordData".xWriteDblExportProdDataBusy, DSTBLK => "DB_ExportProdData".aProdData)
   END_RUNG
   RUNG wire#powerrail
      P_Contact(operand := "DB_FromHmi".xExportProdData, bit := "DB_RecordData".xFP_ExportProdData)
   END_RUNG wire#w1
   // the same network as SCL:
   #_w1 := "DB_FromHmi".xExportProdData AND NOT "DB_RecordData".xFP_ExportProdData;   // rising edge of "DB_FromHmi".xExportProdData
   "DB_RecordData".xFP_ExportProdData := "DB_FromHmi".xExportProdData;
   "DB_RecordData".nWriteDblExportProdDataResult := WRIT_DBL(REQ := #_w1,
                           SRCBLK := "DB_ProductionRecords".aProdData,
                           BUSY => "DB_RecordData".xWriteDblExportProdDataBusy,
                           DSTBLK => "DB_ExportProdData".aProdData);
END_REGION

REGION Network 5: Export DB_ExportProdData as recipe
   RUNG wire#powerrail
      { S7_Templates := "recipe_type := Variant" } "iDB_ExportProdData".RecipeExport(REQ := wire#w1, RECIPE_DB := "DB_ExportProdData".aProdData, DONE => "DB_RecordData".xExportProdDataDone, BUSY => "DB_RecordData".xExportProdDataBusy, ERROR => "DB_RecordData".xExportProdDataError, STATUS => "DB_RecordData".wExportProdDataStatus)
   END_RUNG
   RUNG wire#powerrail
      Contact( "DB_FromHmi".xExportProdData )
      I_Contact( "DB_RecordData".xWriteDblExportProdDataBusy )
   END_RUNG wire#w1
   // the same network as SCL:
   "iDB_ExportProdData"(REQ := "DB_FromHmi".xExportProdData AND NOT "DB_RecordData".xWriteDblExportProdDataBusy,   // RecipeExport
                        RECIPE_DB := "DB_ExportProdData".aProdData,
                        DONE => "DB_RecordData".xExportProdDataDone,
                        BUSY => "DB_RecordData".xExportProdDataBusy,
                        ERROR => "DB_RecordData".xExportProdDataError,
                        STATUS => "DB_RecordData".wExportProdDataStatus);
END_REGION

REGION Network 6: Reset export commande when done
   RUNG wire#powerrail
      Contact( "DB_RecordData".xExportProdDataDone )
      wire#w1
      R_Coil( "DB_FromHmi".xExportProdData )
   END_RUNG
   RUNG wire#powerrail
      Contact( "DB_FromHmi".xResetFault )
   END_RUNG wire#w1
   // the same network as SCL:
   IF "DB_RecordData".xExportProdDataDone OR "DB_FromHmi".xResetFault THEN
       "DB_FromHmi".xExportProdData := FALSE;
   END_IF;
END_REGION

REGION Network 7: Record the error
   RUNG wire#powerrail
      Contact( "DB_RecordData".xExportProdDataError )
      Move(in := "DB_RecordData".wExportProdDataStatus, out1 => "DB_RecordData".wMemExportProdDataStatus)
   END_RUNG
   // the same network as SCL:
   IF "DB_RecordData".xExportProdDataError THEN
       "DB_RecordData".wMemExportProdDataStatus := "DB_RecordData".wExportProdDataStatus;
   END_IF;
END_REGION

REGION Network 8: Copy from DB_ProductionRecords to DB_ExportFlatCtrlRobot1
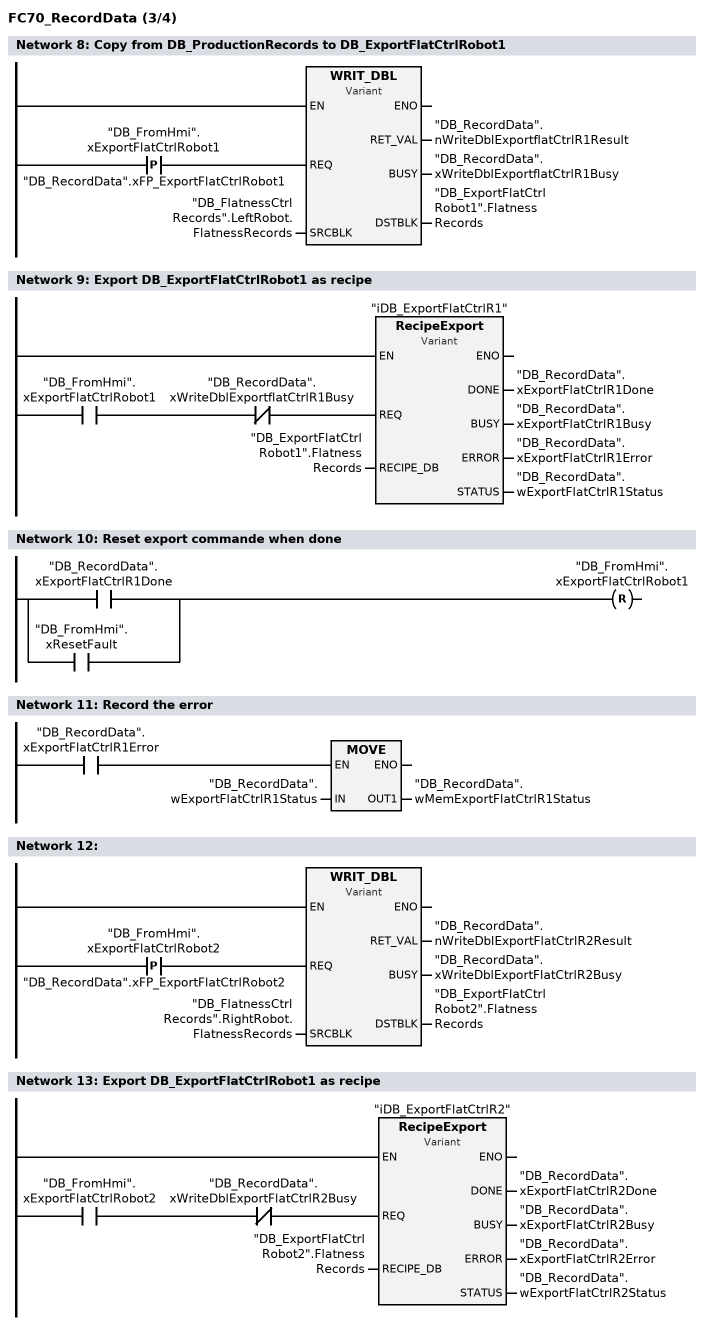
   RUNG wire#powerrail
      { S7_Templates := "[src_type := Variant, dest_type := Variant]" } WRIT_DBL(REQ := wire#w1, SRCBLK := "DB_FlatnessCtrlRecords".LeftRobot.FlatnessRecords, RET_VAL => "DB_RecordData".nWriteDblExportflatCtrlR1Result, BUSY => "DB_RecordData".xWriteDblExportflatCtrlR1Busy, DSTBLK => "DB_ExportFlatCtrlRobot1".FlatnessRecords)
   END_RUNG
   RUNG wire#powerrail
      P_Contact(operand := "DB_FromHmi".xExportFlatCtrlRobot1, bit := "DB_RecordData".xFP_ExportFlatCtrlRobot1)
   END_RUNG wire#w1
   // the same network as SCL:
   #_w1 := "DB_FromHmi".xExportFlatCtrlRobot1 AND NOT "DB_RecordData".xFP_ExportFlatCtrlRobot1;   // rising edge of "DB_FromHmi".xExportFlatCtrlRobot1
   "DB_RecordData".xFP_ExportFlatCtrlRobot1 := "DB_FromHmi".xExportFlatCtrlRobot1;
   "DB_RecordData".nWriteDblExportflatCtrlR1Result := WRIT_DBL(REQ := #_w1,
                           SRCBLK := "DB_FlatnessCtrlRecords".LeftRobot.FlatnessRecords,
                           BUSY => "DB_RecordData".xWriteDblExportflatCtrlR1Busy,
                           DSTBLK => "DB_ExportFlatCtrlRobot1".FlatnessRecords);
END_REGION

REGION Network 9: Export DB_ExportFlatCtrlRobot1 as recipe
   RUNG wire#powerrail
      { S7_Templates := "recipe_type := Variant" } "iDB_ExportFlatCtrlR1".RecipeExport(REQ := wire#w1, RECIPE_DB := "DB_ExportFlatCtrlRobot1".FlatnessRecords, DONE => "DB_RecordData".xExportFlatCtrlR1Done, BUSY => "DB_RecordData".xExportFlatCtrlR1Busy, ERROR => "DB_RecordData".xExportFlatCtrlR1Error, STATUS => "DB_RecordData".wExportFlatCtrlR1Status)
   END_RUNG
   RUNG wire#powerrail
      Contact( "DB_FromHmi".xExportFlatCtrlRobot1 )
      I_Contact( "DB_RecordData".xWriteDblExportflatCtrlR1Busy )
   END_RUNG wire#w1
   // the same network as SCL:
   "iDB_ExportFlatCtrlR1"(REQ := "DB_FromHmi".xExportFlatCtrlRobot1 AND NOT "DB_RecordData".xWriteDblExportflatCtrlR1Busy,   // RecipeExport
                          RECIPE_DB := "DB_ExportFlatCtrlRobot1".FlatnessRecords,
                          DONE => "DB_RecordData".xExportFlatCtrlR1Done,
                          BUSY => "DB_RecordData".xExportFlatCtrlR1Busy,
                          ERROR => "DB_RecordData".xExportFlatCtrlR1Error,
                          STATUS => "DB_RecordData".wExportFlatCtrlR1Status);
END_REGION

REGION Network 10: Reset export commande when done
   RUNG wire#powerrail
      Contact( "DB_RecordData".xExportFlatCtrlR1Done )
      wire#w1
      R_Coil( "DB_FromHmi".xExportFlatCtrlRobot1 )
   END_RUNG
   RUNG wire#powerrail
      Contact( "DB_FromHmi".xResetFault )
   END_RUNG wire#w1
   // the same network as SCL:
   IF "DB_RecordData".xExportFlatCtrlR1Done OR "DB_FromHmi".xResetFault THEN
       "DB_FromHmi".xExportFlatCtrlRobot1 := FALSE;
   END_IF;
END_REGION

REGION Network 11: Record the error
   RUNG wire#powerrail
      Contact( "DB_RecordData".xExportFlatCtrlR1Error )
      Move(in := "DB_RecordData".wExportFlatCtrlR1Status, out1 => "DB_RecordData".wMemExportFlatCtrlR1Status)
   END_RUNG
   // the same network as SCL:
   IF "DB_RecordData".xExportFlatCtrlR1Error THEN
       "DB_RecordData".wMemExportFlatCtrlR1Status := "DB_RecordData".wExportFlatCtrlR1Status;
   END_IF;
END_REGION

REGION Network 12
   RUNG wire#powerrail
      { S7_Templates := "[src_type := Variant, dest_type := Variant]" } WRIT_DBL(REQ := wire#w1, SRCBLK := "DB_FlatnessCtrlRecords".RightRobot.FlatnessRecords, RET_VAL => "DB_RecordData".nWriteDblExportFlatCtrlR2Result, BUSY => "DB_RecordData".xWriteDblExportFlatCtrlR2Busy, DSTBLK => "DB_ExportFlatCtrlRobot2".FlatnessRecords)
   END_RUNG
   RUNG wire#powerrail
      P_Contact(operand := "DB_FromHmi".xExportFlatCtrlRobot2, bit := "DB_RecordData".xFP_ExportFlatCtrlRobot2)
   END_RUNG wire#w1
   // the same network as SCL:
   #_w1 := "DB_FromHmi".xExportFlatCtrlRobot2 AND NOT "DB_RecordData".xFP_ExportFlatCtrlRobot2;   // rising edge of "DB_FromHmi".xExportFlatCtrlRobot2
   "DB_RecordData".xFP_ExportFlatCtrlRobot2 := "DB_FromHmi".xExportFlatCtrlRobot2;
   "DB_RecordData".nWriteDblExportFlatCtrlR2Result := WRIT_DBL(REQ := #_w1,
                           SRCBLK := "DB_FlatnessCtrlRecords".RightRobot.FlatnessRecords,
                           BUSY => "DB_RecordData".xWriteDblExportFlatCtrlR2Busy,
                           DSTBLK => "DB_ExportFlatCtrlRobot2".FlatnessRecords);
END_REGION

REGION Network 13: Export DB_ExportFlatCtrlRobot1 as recipe
   RUNG wire#powerrail
      { S7_Templates := "recipe_type := Variant" } "iDB_ExportFlatCtrlR2".RecipeExport(REQ := wire#w1, RECIPE_DB := "DB_ExportFlatCtrlRobot2".FlatnessRecords, DONE => "DB_RecordData".xExportFlatCtrlR2Done, BUSY => "DB_RecordData".xExportFlatCtrlR2Busy, ERROR => "DB_RecordData".xExportFlatCtrlR2Error, STATUS => "DB_RecordData".wExportFlatCtrlR2Status)
   END_RUNG
   RUNG wire#powerrail
      Contact( "DB_FromHmi".xExportFlatCtrlRobot2 )
      I_Contact( "DB_RecordData".xWriteDblExportFlatCtrlR2Busy )
   END_RUNG wire#w1
   // the same network as SCL:
   "iDB_ExportFlatCtrlR2"(REQ := "DB_FromHmi".xExportFlatCtrlRobot2 AND NOT "DB_RecordData".xWriteDblExportFlatCtrlR2Busy,   // RecipeExport
                          RECIPE_DB := "DB_ExportFlatCtrlRobot2".FlatnessRecords,
                          DONE => "DB_RecordData".xExportFlatCtrlR2Done,
                          BUSY => "DB_RecordData".xExportFlatCtrlR2Busy,
                          ERROR => "DB_RecordData".xExportFlatCtrlR2Error,
                          STATUS => "DB_RecordData".wExportFlatCtrlR2Status);
END_REGION

REGION Network 14: Reset export commande when done
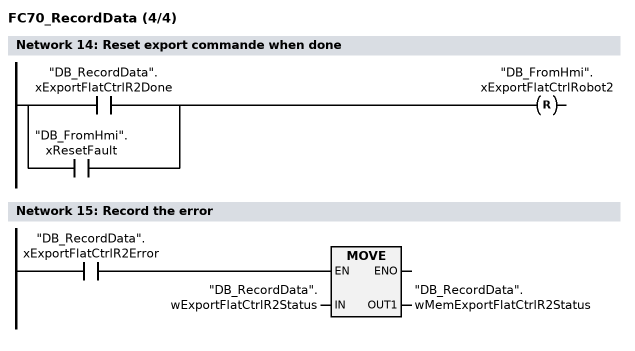
   RUNG wire#powerrail
      Contact( "DB_RecordData".xExportFlatCtrlR2Done )
      wire#w1
      R_Coil( "DB_FromHmi".xExportFlatCtrlRobot2 )
   END_RUNG
   RUNG wire#powerrail
      Contact( "DB_FromHmi".xResetFault )
   END_RUNG wire#w1
   // the same network as SCL:
   IF "DB_RecordData".xExportFlatCtrlR2Done OR "DB_FromHmi".xResetFault THEN
       "DB_FromHmi".xExportFlatCtrlRobot2 := FALSE;
   END_IF;
END_REGION

REGION Network 15: Record the error
   RUNG wire#powerrail
      Contact( "DB_RecordData".xExportFlatCtrlR2Error )
      Move(in := "DB_RecordData".wExportFlatCtrlR2Status, out1 => "DB_RecordData".wMemExportFlatCtrlR2Status)
   END_RUNG
   // the same network as SCL:
   IF "DB_RecordData".xExportFlatCtrlR2Error THEN
       "DB_RecordData".wMemExportFlatCtrlR2Status := "DB_RecordData".wExportFlatCtrlR2Status;
   END_IF;
END_REGION
END_FUNCTION

FUNCTION_BLOCK "FB70_ProductionRecord"
{ S7_Optimized_Access := 'TRUE' }
VERSION : 0.1
   VAR_INPUT 
      usiCurrentLayerType { ExternalAccessible := 'False'; ExternalVisible := 'False'; ExternalWritable := 'False'} : USInt;
      uiCbsNumber { ExternalAccessible := 'False'; ExternalVisible := 'False'; ExternalWritable := 'False'} : UInt;
      uiCurrentJobNumberRobot1 { ExternalAccessible := 'False'; ExternalVisible := 'False'; ExternalWritable := 'False'} : UInt;
      uiCurrentJobNumberRobot2 { ExternalAccessible := 'False'; ExternalVisible := 'False'; ExternalWritable := 'False'} : UInt;
      uiPaperUsedRobot1 { ExternalAccessible := 'False'; ExternalVisible := 'False'; ExternalWritable := 'False'} : UInt;
      uiPaperUsedRobot2 { ExternalAccessible := 'False'; ExternalVisible := 'False'; ExternalWritable := 'False'} : UInt;
      WorkRecipe { ExternalAccessible := 'False'; ExternalVisible := 'False'; ExternalWritable := 'False'} : "stWorkRecipe";
   END_VAR

   VAR_OUTPUT 
      uiRecordMax { ExternalAccessible := 'False'; ExternalVisible := 'False'; ExternalWritable := 'False'} : UInt;
      uiRecordMin { ExternalAccessible := 'False'; ExternalVisible := 'False'; ExternalWritable := 'False'} : UInt;
      uiNbrDisplyedLine { ExternalAccessible := 'False'; ExternalVisible := 'False'; ExternalWritable := 'False'} : UInt;   // Number of displayed lime of production
      uiFirstRecordDisplayed { ExternalAccessible := 'False'; ExternalVisible := 'False'; ExternalWritable := 'False'} : UInt;   // First record displayed
      uiLastRecordDisplayed { ExternalAccessible := 'False'; ExternalVisible := 'False'; ExternalWritable := 'False'} : UInt;   // Last record displayed
      aDisplayProdData { ExternalAccessible := 'False'; ExternalVisible := 'False'; ExternalWritable := 'False'} : Array[0..9] of "stProductionRecord";
   END_VAR

